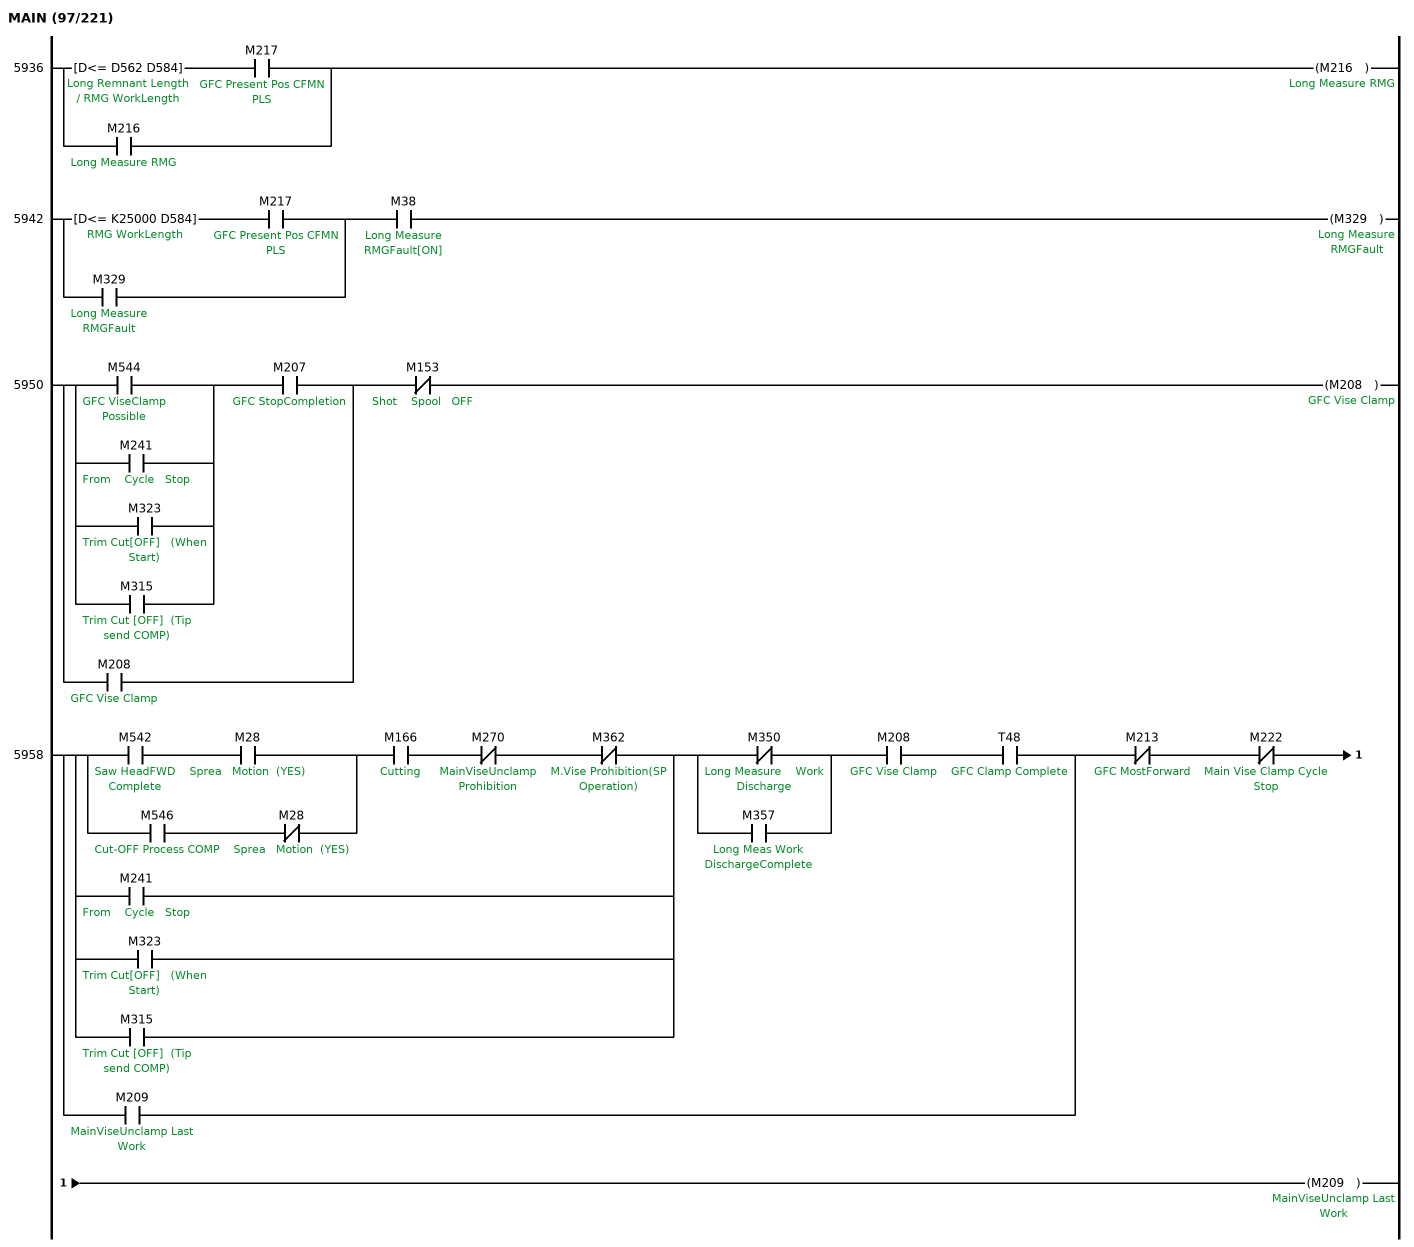
[picture p96: ladder of MAIN, rungs at steps 5936 to 5958]
5936  LDD<=   D562 D584  ; Long Remnant Length / RMG WorkLength
      AND     M217  ; GFC Present Pos CFMN PLS
      OR      M216  ; Long Measure RMG
      OUT     M216  ; Long Measure RMG
5942  LDD<=   K25000 D584  ; RMG WorkLength
      AND     M217  ; GFC Present Pos CFMN PLS
      OR      M329  ; Long Measure RMGFault
      AND     M38  ; Long Measure RMGFault[ON]
      OUT     M329  ; Long Measure RMGFault
5950  LD      M544  ; GFC ViseClamp   Possible
      OR      M241  ; From    Cycle   Stop
      OR      M323  ; Trim Cut[OFF]   (When   Start)
      OR      M315  ; Trim Cut [OFF]  (Tip send COMP)
      AND     M207  ; GFC StopCompletion
      OR      M208  ; GFC Vise Clamp
      ANI     M153  ; Shot    Spool   OFF
      OUT     M208  ; GFC Vise Clamp
5958  LD      M542  ; Saw HeadFWD     Complete
      AND     M28  ; Sprea   Motion  (YES)
      LD      M546  ; Cut-OFF Process COMP
      ANI     M28  ; Sprea   Motion  (YES)
      ORB
      AND     M166  ; Cutting
      ANI     M270  ; MainViseUnclamp Prohibition
      ANI     M362  ; M.Vise Prohibition(SP Operation)
      OR      M241  ; From    Cycle   Stop
      OR      M323  ; Trim Cut[OFF]   (When   Start)
      OR      M315  ; Trim Cut [OFF]  (Tip send COMP)
      LDI     M350  ; Long Measure    Work Discharge
      OR      M357  ; Long Meas Work DischargeComplete
      ANB
      AND     M208  ; GFC Vise Clamp
      AND     T48  ; GFC Clamp Complete
      OR      M209  ; MainViseUnclamp Last    Work
      ANI     M213  ; GFC MostForward
      ANI     M222  ; Main Vise Clamp Cycle Stop
      OUT     M209  ; MainViseUnclamp Last    Work
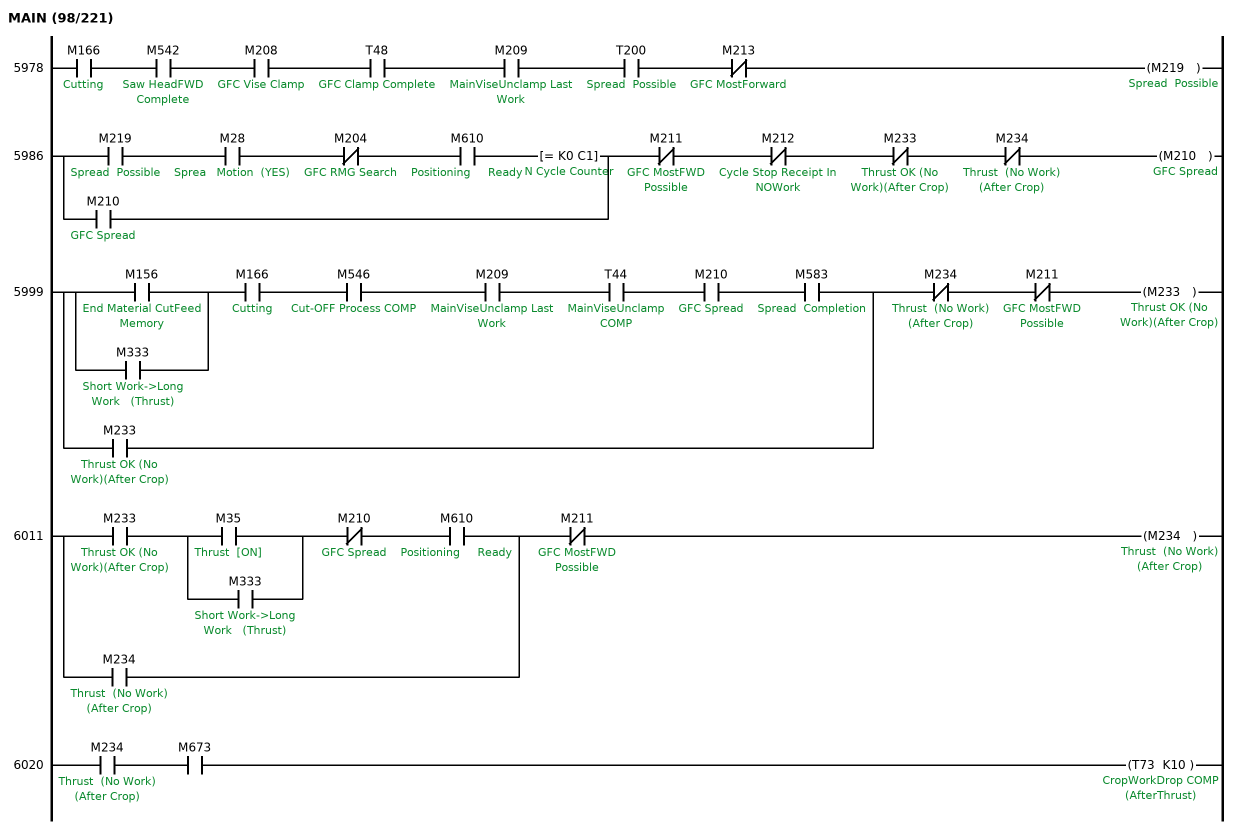
5978  LD      M166  ; Cutting
      AND     M542  ; Saw HeadFWD     Complete
      AND     M208  ; GFC Vise Clamp
      AND     T48  ; GFC Clamp Complete
      AND     M209  ; MainViseUnclamp Last    Work
      AND     T200  ; Spread  Possible
      ANI     M213  ; GFC MostForward
      OUT     M219  ; Spread  Possible
5986  LD      M219  ; Spread  Possible
      AND     M28  ; Sprea   Motion  (YES)
      ANI     M204  ; GFC RMG Search
      AND     M610  ; Positioning     Ready
      AND=    K0 C1  ; N Cycle Counter
      OR      M210  ; GFC Spread
      ANI     M211  ; GFC MostFWD     Possible
      ANI     M212  ; Cycle Stop Receipt In NOWork
      ANI     M233  ; Thrust OK (No Work)(After Crop)
      ANI     M234  ; Thrust  (No Work) (After Crop)
      OUT     M210  ; GFC Spread
5999  LD      M156  ; End Material CutFeed Memory
      OR      M333  ; Short Work->Long Work   (Thrust)
      AND     M166  ; Cutting
      AND     M546  ; Cut-OFF Process COMP
      AND     M209  ; MainViseUnclamp Last    Work
      AND     T44  ; MainViseUnclamp COMP
      AND     M210  ; GFC Spread
      AND     M583  ; Spread  Completion
      OR      M233  ; Thrust OK (No Work)(After Crop)
      ANI     M234  ; Thrust  (No Work) (After Crop)
      ANI     M211  ; GFC MostFWD     Possible
      OUT     M233  ; Thrust OK (No Work)(After Crop)
6011  LD      M233  ; Thrust OK (No Work)(After Crop)
      LD      M35  ; Thrust  [ON]
      OR      M333  ; Short Work->Long Work   (Thrust)
      ANB
      ANI     M210  ; GFC Spread
      AND     M610  ; Positioning     Ready
      OR      M234  ; Thrust  (No Work) (After Crop)
      ANI     M211  ; GFC MostFWD     Possible
      OUT     M234  ; Thrust  (No Work) (After Crop)
6020  LD      M234  ; Thrust  (No Work) (After Crop)
      AND     M673
      OUT     T73 K10  ; CropWorkDrop COMP (AfterThrust)
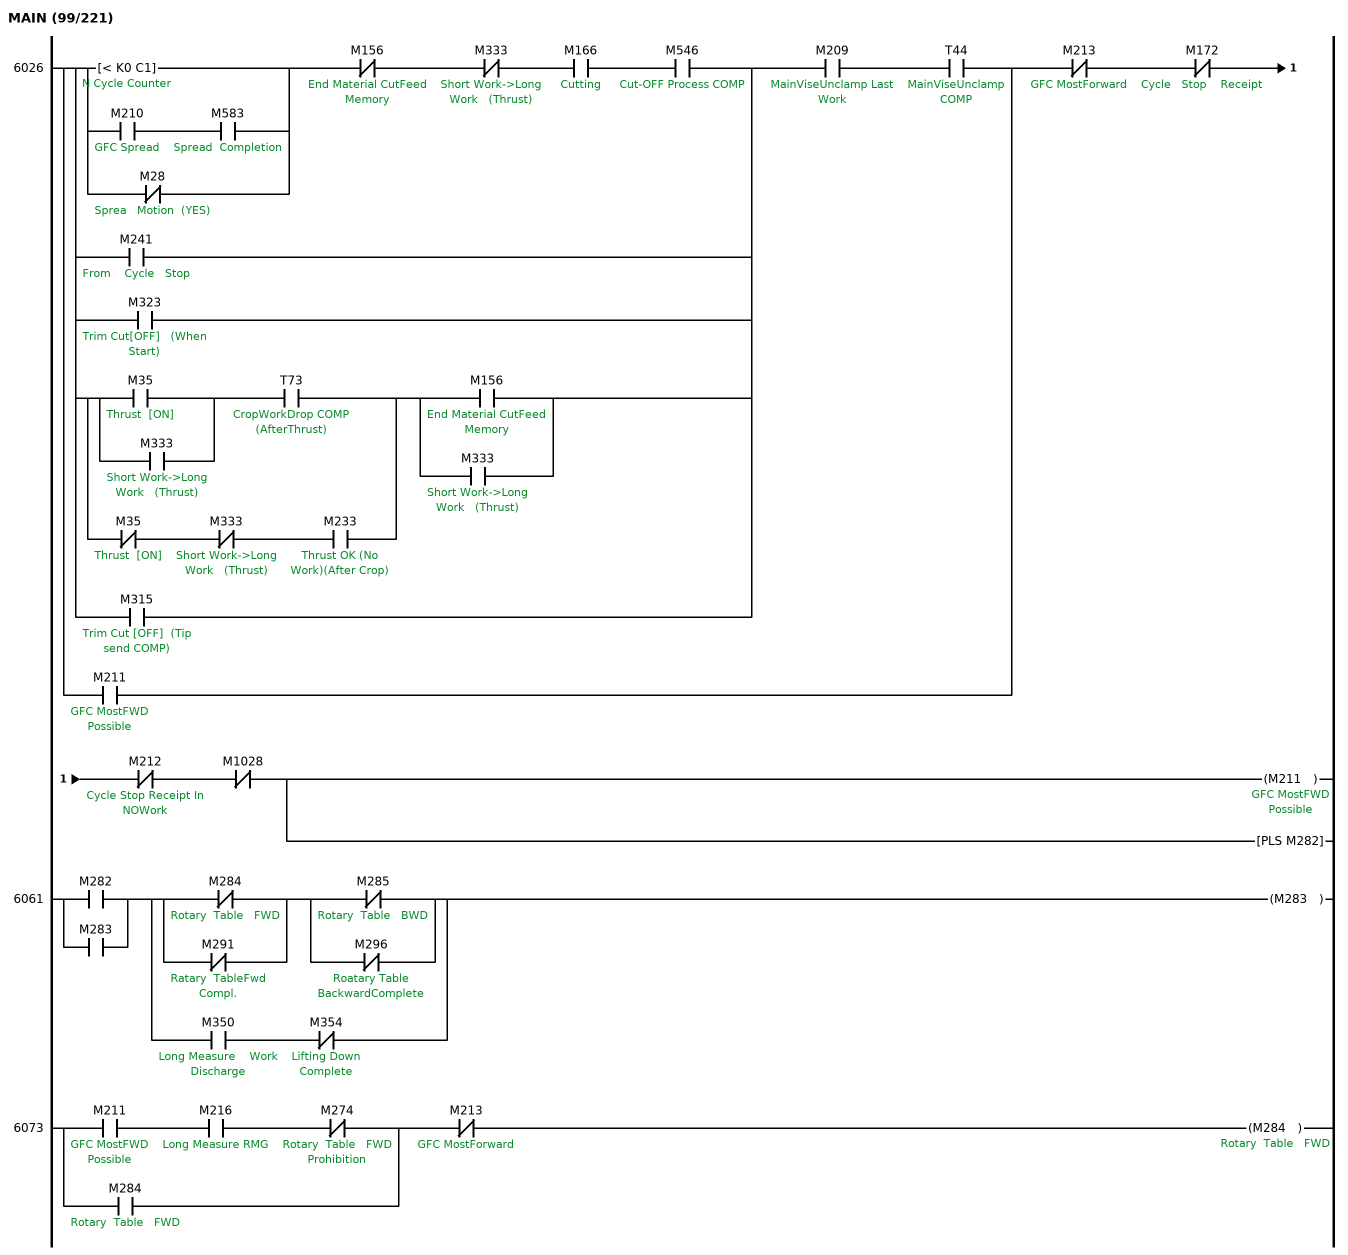
6026  LD<     K0 C1  ; N Cycle Counter
      LD      M210  ; GFC Spread
      AND     M583  ; Spread  Completion
      ORB
      ORI     M28  ; Sprea   Motion  (YES)
      ANI     M156  ; End Material CutFeed Memory
      ANI     M333  ; Short Work->Long Work   (Thrust)
      AND     M166  ; Cutting
      AND     M546  ; Cut-OFF Process COMP
      OR      M241  ; From    Cycle   Stop
      OR      M323  ; Trim Cut[OFF]   (When   Start)
      LD      M35  ; Thrust  [ON]
      OR      M333  ; Short Work->Long Work   (Thrust)
      AND     T73  ; CropWorkDrop COMP (AfterThrust)
      LDI     M35  ; Thrust  [ON]
      ANI     M333  ; Short Work->Long Work   (Thrust)
      AND     M233  ; Thrust OK (No Work)(After Crop)
      ORB
      LD      M156  ; End Material CutFeed Memory
      OR      M333  ; Short Work->Long Work   (Thrust)
      ANB
      ORB
      OR      M315  ; Trim Cut [OFF]  (Tip send COMP)
      AND     M209  ; MainViseUnclamp Last    Work
      AND     T44  ; MainViseUnclamp COMP
      OR      M211  ; GFC MostFWD     Possible
      ANI     M213  ; GFC MostForward
      ANI     M172  ; Cycle   Stop    Receipt
      ANI     M212  ; Cycle Stop Receipt In NOWork
      ANI     M1028
      OUT     M211  ; GFC MostFWD     Possible
      PLS     M282
6061  LD      M282
      OR      M283
      LDI     M284  ; Rotary  Table   FWD
      ORI     M291  ; Ratary  TableFwd Compl.
      LDI     M285  ; Rotary  Table   BWD
      ORI     M296  ; Roatary Table   BackwardComplete
      ANB
      LD      M350  ; Long Measure    Work Discharge
      ANI     M354  ; Lifting Down    Complete
      ORB
      ANB
      OUT     M283
6073  LD      M211  ; GFC MostFWD     Possible
      AND     M216  ; Long Measure RMG
      ANI     M274  ; Rotary  Table   FWD Prohibition
      OR      M284  ; Rotary  Table   FWD
      ANI     M213  ; GFC MostForward
      OUT     M284  ; Rotary  Table   FWD
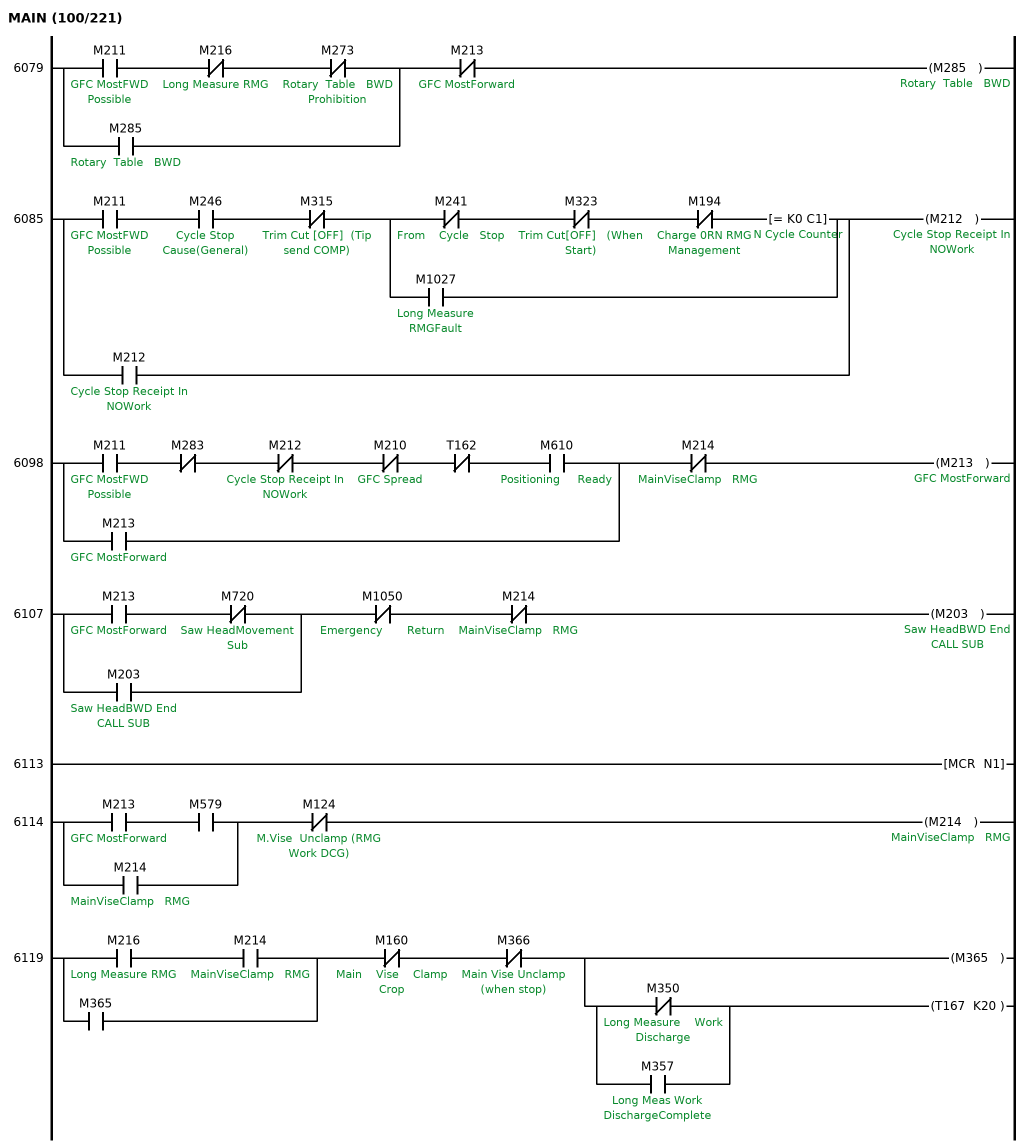
6079  LD      M211  ; GFC MostFWD     Possible
      ANI     M216  ; Long Measure RMG
      ANI     M273  ; Rotary  Table   BWD Prohibition
      OR      M285  ; Rotary  Table   BWD
      ANI     M213  ; GFC MostForward
      OUT     M285  ; Rotary  Table   BWD
6085  LD      M211  ; GFC MostFWD     Possible
      AND     M246  ; Cycle Stop Cause(General)
      ANI     M315  ; Trim Cut [OFF]  (Tip send COMP)
      LDI     M241  ; From    Cycle   Stop
      ANI     M323  ; Trim Cut[OFF]   (When   Start)
      ANI     M194  ; Charge 0RN RMG  Management
      AND=    K0 C1  ; N Cycle Counter
      OR      M1027  ; Long Measure RMGFault
      ANB
      OR      M212  ; Cycle Stop Receipt In NOWork
      OUT     M212  ; Cycle Stop Receipt In NOWork
6098  LD      M211  ; GFC MostFWD     Possible
      ANI     M283
      ANI     M212  ; Cycle Stop Receipt In NOWork
      ANI     M210  ; GFC Spread
      ANI     T162
      AND     M610  ; Positioning     Ready
      OR      M213  ; GFC MostForward
      ANI     M214  ; MainViseClamp   RMG
      OUT     M213  ; GFC MostForward
6107  LD      M213  ; GFC MostForward
      ANI     M720  ; Saw HeadMovementSub
      OR      M203  ; Saw HeadBWD End CALL SUB
      ANI     M1050  ; Emergency       Return
      ANI     M214  ; MainViseClamp   RMG
      OUT     M203  ; Saw HeadBWD End CALL SUB
6113  MCR     N1
6114  LD      M213  ; GFC MostForward
      AND     M579
      OR      M214  ; MainViseClamp   RMG
      ANI     M124  ; M.Vise  Unclamp (RMG Work DCG)
      OUT     M214  ; MainViseClamp   RMG
6119  LD      M216  ; Long Measure RMG
      AND     M214  ; MainViseClamp   RMG
      OR      M365
      ANI     M160  ; Main    Vise    Clamp   Crop
      ANI     M366  ; Main Vise Unclamp (when stop)
      OUT     M365
      LDI     M350  ; Long Measure    Work Discharge
      OR      M357  ; Long Meas Work DischargeComplete
      ANB
      OUT     T167 K20
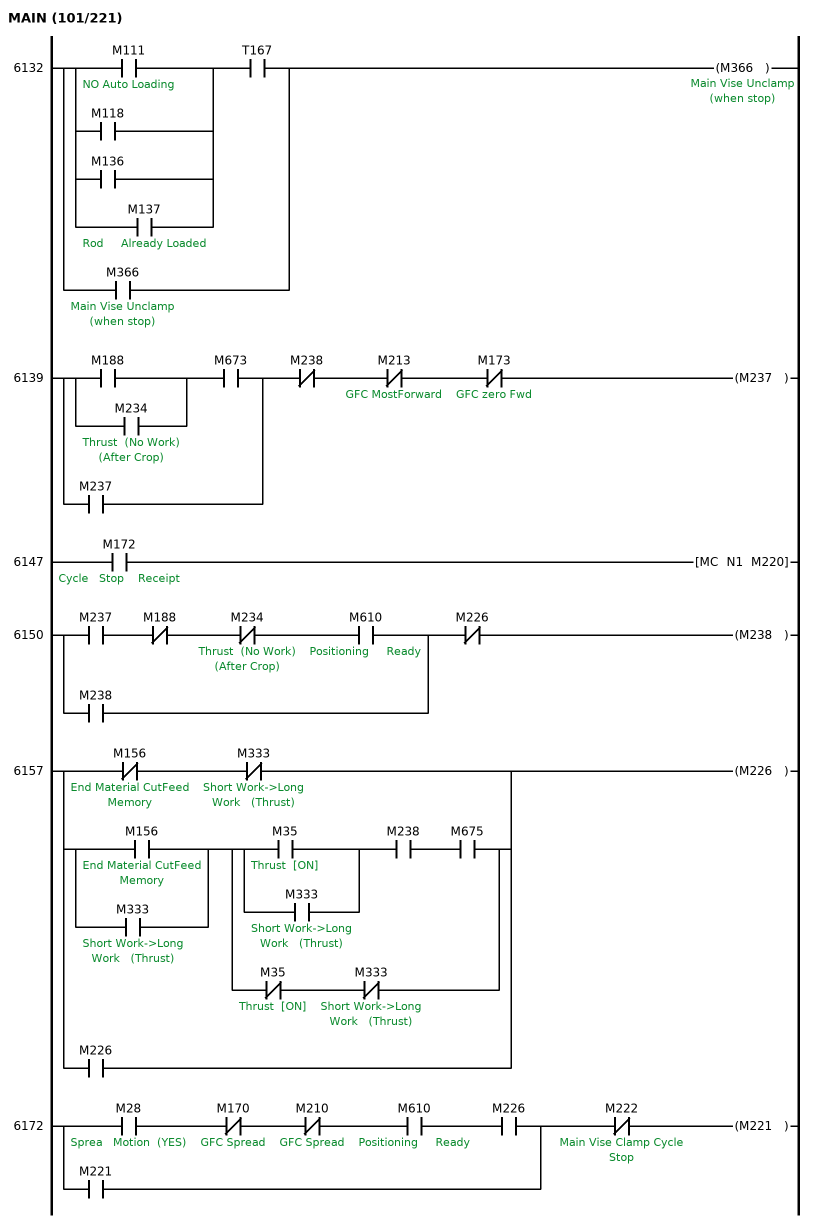
6132  LD      M111  ; NO Auto Loading
      OR      M118
      OR      M136
      OR      M137  ; Rod     Already Loaded
      AND     T167
      OR      M366  ; Main Vise Unclamp (when stop)
      OUT     M366  ; Main Vise Unclamp (when stop)
6139  LD      M188
      OR      M234  ; Thrust  (No Work) (After Crop)
      AND     M673
      OR      M237
      ANI     M238
      ANI     M213  ; GFC MostForward
      ANI     M173  ; GFC zero Fwd
      OUT     M237
6147  LD      M172  ; Cycle   Stop    Receipt
      MC      N1 M220
6150  LD      M237
      ANI     M188
      ANI     M234  ; Thrust  (No Work) (After Crop)
      AND     M610  ; Positioning     Ready
      OR      M238
      ANI     M226
      OUT     M238
6157  LDI     M156  ; End Material CutFeed Memory
      ANI     M333  ; Short Work->Long Work   (Thrust)
      LD      M156  ; End Material CutFeed Memory
      OR      M333  ; Short Work->Long Work   (Thrust)
      LD      M35  ; Thrust  [ON]
      OR      M333  ; Short Work->Long Work   (Thrust)
      AND     M238
      AND     M675
      LDI     M35  ; Thrust  [ON]
      ANI     M333  ; Short Work->Long Work   (Thrust)
      ORB
      ANB
      ORB
      OR      M226
      OUT     M226
6172  LD      M28  ; Sprea   Motion  (YES)
      ANI     M170  ; GFC Spread
      ANI     M210  ; GFC Spread
      AND     M610  ; Positioning     Ready
      AND     M226
      OR      M221
      ANI     M222  ; Main Vise Clamp Cycle Stop
      OUT     M221
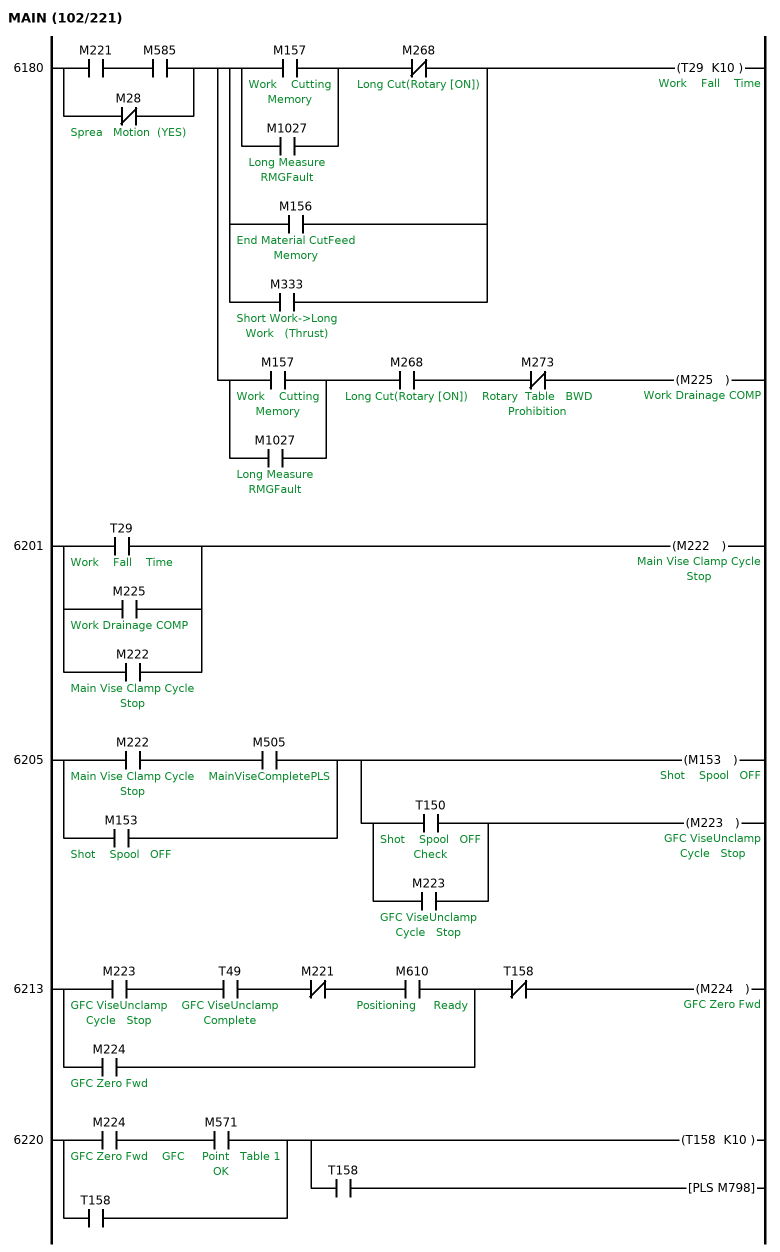
6180  LD      M221
      AND     M585
      ORI     M28  ; Sprea   Motion  (YES)
      MPS
      LD      M157  ; Work    Cutting Memory
      OR      M1027  ; Long Measure RMGFault
      ANI     M268  ; Long Cut(Rotary [ON])
      OR      M156  ; End Material CutFeed Memory
      OR      M333  ; Short Work->Long Work   (Thrust)
      ANB
      OUT     T29 K10  ; Work    Fall    Time
      MPP
      LD      M157  ; Work    Cutting Memory
      OR      M1027  ; Long Measure RMGFault
      ANB
      AND     M268  ; Long Cut(Rotary [ON])
      ANI     M273  ; Rotary  Table   BWD Prohibition
      OUT     M225  ; Work Drainage COMP
6201  LD      T29  ; Work    Fall    Time
      OR      M225  ; Work Drainage COMP
      OR      M222  ; Main Vise Clamp Cycle Stop
      OUT     M222  ; Main Vise Clamp Cycle Stop
6205  LD      M222  ; Main Vise Clamp Cycle Stop
      AND     M505  ; MainViseCompletePLS
      OR      M153  ; Shot    Spool   OFF
      OUT     M153  ; Shot    Spool   OFF
      LD      T150  ; Shot    Spool   OFF     Check
      OR      M223  ; GFC ViseUnclamp Cycle   Stop
      ANB
      OUT     M223  ; GFC ViseUnclamp Cycle   Stop
6213  LD      M223  ; GFC ViseUnclamp Cycle   Stop
      AND     T49  ; GFC ViseUnclamp Complete
      ANI     M221
      AND     M610  ; Positioning     Ready
      OR      M224  ; GFC Zero Fwd
      ANI     T158
      OUT     M224  ; GFC Zero Fwd
6220  LD      M224  ; GFC Zero Fwd
      AND     M571  ; GFC     Point   Table 1 OK
      OR      T158
      OUT     T158 K10
      AND     T158
      PLS     M798
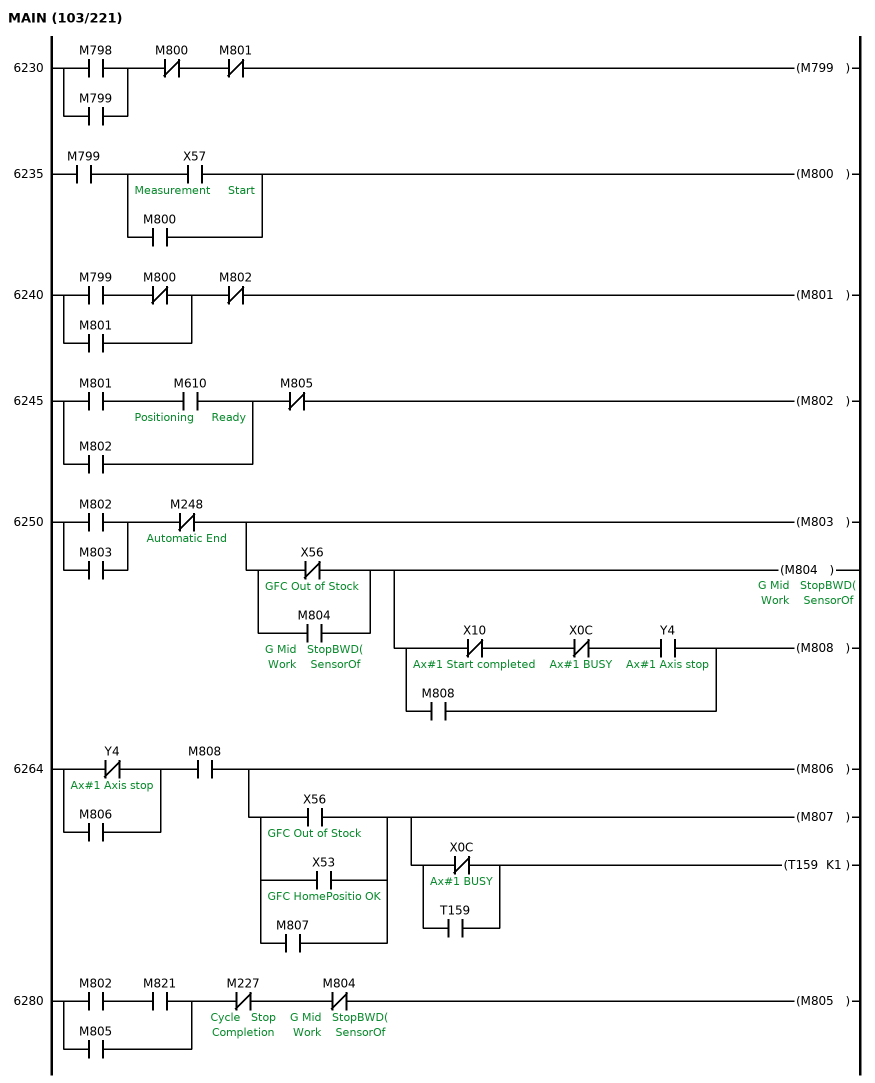
6230  LD      M798
      OR      M799
      ANI     M800
      ANI     M801
      OUT     M799
6235  LD      M799
      LD      X57  ; Measurement     Start
      OR      M800
      ANB
      OUT     M800
6240  LD      M799
      ANI     M800
      OR      M801
      ANI     M802
      OUT     M801
6245  LD      M801
      AND     M610  ; Positioning     Ready
      OR      M802
      ANI     M805
      OUT     M802
6250  LD      M802
      OR      M803
      ANI     M248  ; Automatic End
      OUT     M803
      LDI     X56  ; GFC Out of Stock
      OR      M804  ; G Mid   StopBWD(Work    SensorOf
      ANB
      OUT     M804  ; G Mid   StopBWD(Work    SensorOf
      LDI     X10  ; Ax#1 Start completed
      ANI     X0C  ; Ax#1 BUSY
      AND     Y4  ; Ax#1 Axis stop
      OR      M808
      ANB
      OUT     M808
6264  LDI     Y4  ; Ax#1 Axis stop
      OR      M806
      AND     M808
      OUT     M806
      LD      X56  ; GFC Out of Stock
      OR      X53  ; GFC HomePositio OK
      OR      M807
      ANB
      OUT     M807
      LDI     X0C  ; Ax#1 BUSY
      OR      T159
      ANB
      OUT     T159 K1
6280  LD      M802
      AND     M821
      OR      M805
      ANI     M227  ; Cycle   Stop    Completion
      ANI     M804  ; G Mid   StopBWD(Work    SensorOf
      OUT     M805
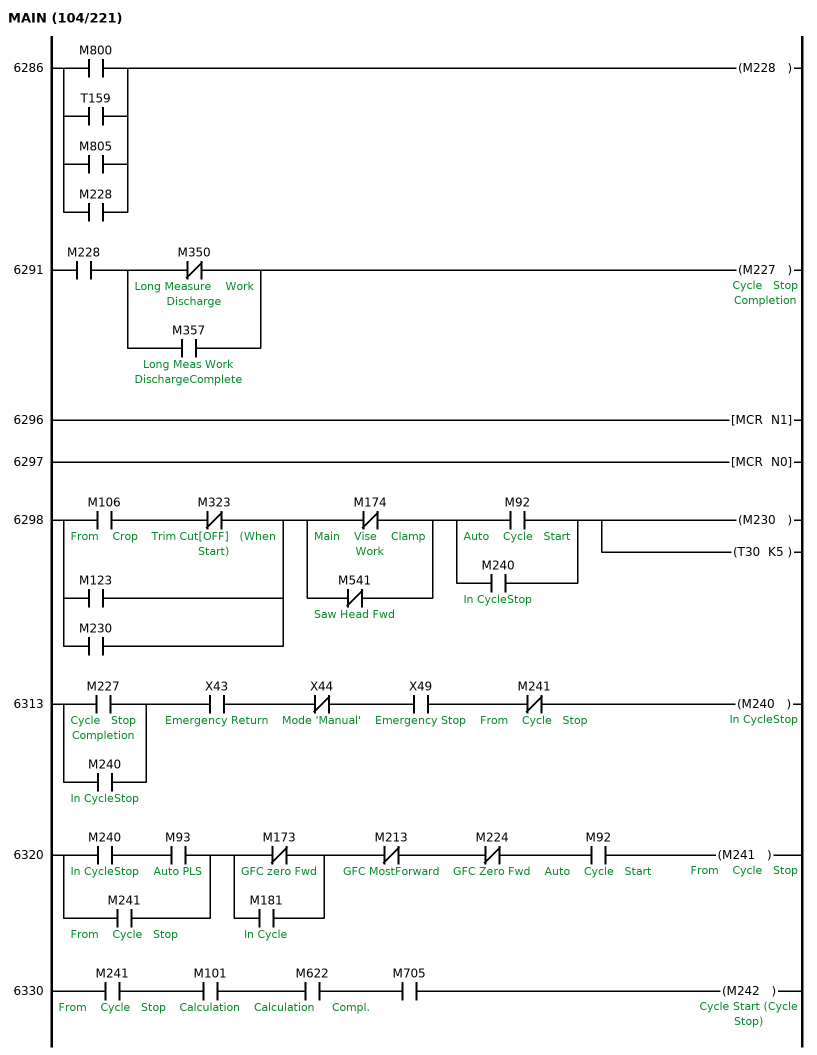
6286  LD      M800
      OR      T159
      OR      M805
      OR      M228
      OUT     M228
6291  LD      M228
      LDI     M350  ; Long Measure    Work Discharge
      OR      M357  ; Long Meas Work DischargeComplete
      ANB
      OUT     M227  ; Cycle   Stop    Completion
6296  MCR     N1
6297  MCR     N0
6298  LD      M106  ; From    Crop
      ANI     M323  ; Trim Cut[OFF]   (When   Start)
      OR      M123
      OR      M230
      LDI     M174  ; Main    Vise    Clamp   Work
      ORI     M541  ; Saw Head Fwd
      ANB
      LD      M92  ; Auto    Cycle   Start
      OR      M240  ; In CycleStop
      ANB
      OUT     M230
      OUT     T30 K5
6313  LD      M227  ; Cycle   Stop    Completion
      OR      M240  ; In CycleStop
      AND     X43  ; Emergency Return
      ANI     X44  ; Mode 'Manual'
      AND     X49  ; Emergency Stop
      ANI     M241  ; From    Cycle   Stop
      OUT     M240  ; In CycleStop
6320  LD      M240  ; In CycleStop
      AND     M93  ; Auto PLS
      OR      M241  ; From    Cycle   Stop
      LDI     M173  ; GFC zero Fwd
      OR      M181  ; In Cycle
      ANB
      ANI     M213  ; GFC MostForward
      ANI     M224  ; GFC Zero Fwd
      AND     M92  ; Auto    Cycle   Start
      OUT     M241  ; From    Cycle   Stop
6330  LD      M241  ; From    Cycle   Stop
      AND     M101  ; Calculation
      AND     M622  ; Calculation     Compl.
      AND     M705
      OUT     M242  ; Cycle Start (Cycle Stop)
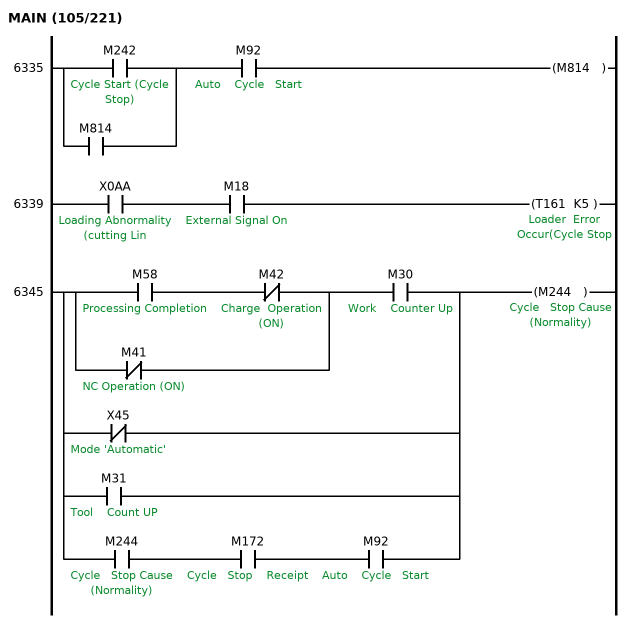
6335  LD      M242  ; Cycle Start (Cycle Stop)
      OR      M814
      AND     M92  ; Auto    Cycle   Start
      OUT     M814
6339  LD      X0AA  ; Loading Abnormality (cutting Lin
      AND     M18  ; External Signal On
      OUT     T161 K5  ; Loader  Error   Occur(Cycle Stop
6345  LD      M58  ; Processing Completion
      ANI     M42  ; Charge  Operation (ON)
      ORI     M41  ; NC Operation (ON)
      AND     M30  ; Work    Counter Up
      ORI     X45  ; Mode 'Automatic'
      OR      M31  ; Tool    Count UP
      LD      M244  ; Cycle   Stop Cause (Normality)
      AND     M172  ; Cycle   Stop    Receipt
      AND     M92  ; Auto    Cycle   Start
      ORB
      OUT     M244  ; Cycle   Stop Cause (Normality)
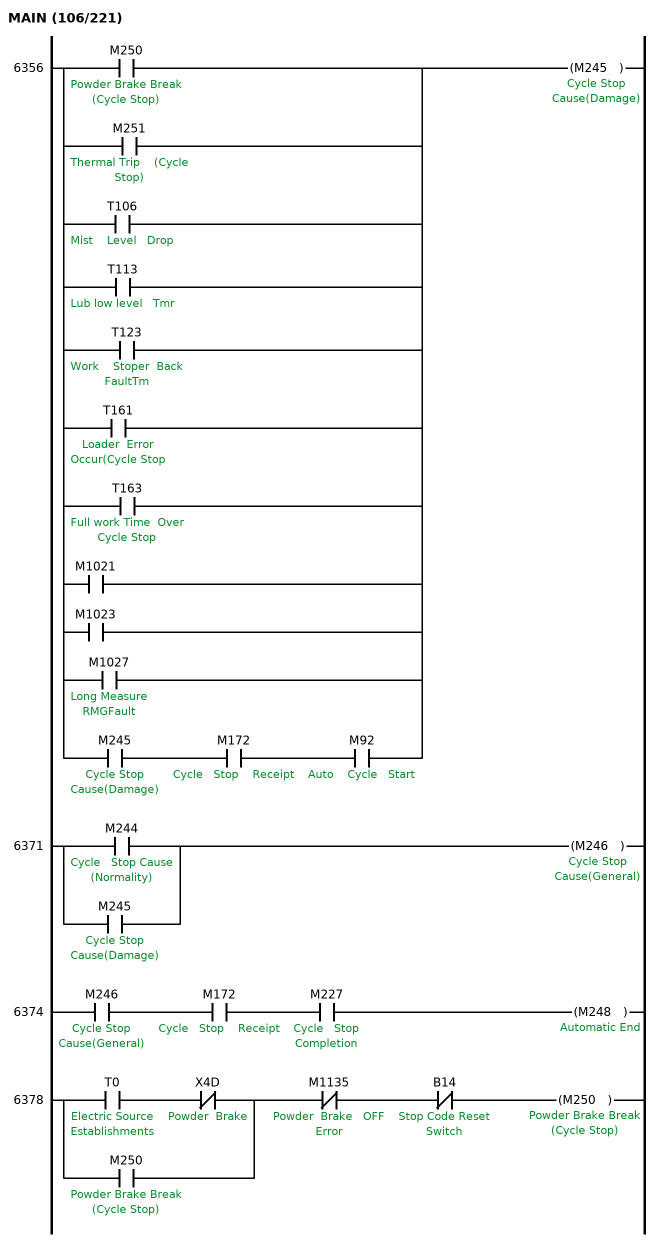
6356  LD      M250  ; Powder Brake Break (Cycle Stop)
      OR      M251  ; Thermal Trip    (Cycle  Stop)
      OR      T106  ; Mist    Level   Drop
      OR      T113  ; Lub low level   Tmr
      OR      T123  ; Work    Stoper  Back    FaultTm
      OR      T161  ; Loader  Error   Occur(Cycle Stop
      OR      T163  ; Full work Time  Over Cycle Stop
      OR      M1021
      OR      M1023
      OR      M1027  ; Long Measure RMGFault
      LD      M245  ; Cycle Stop Cause(Damage)
      AND     M172  ; Cycle   Stop    Receipt
      AND     M92  ; Auto    Cycle   Start
      ORB
      OUT     M245  ; Cycle Stop Cause(Damage)
6371  LD      M244  ; Cycle   Stop Cause (Normality)
      OR      M245  ; Cycle Stop Cause(Damage)
      OUT     M246  ; Cycle Stop Cause(General)
6374  LD      M246  ; Cycle Stop Cause(General)
      AND     M172  ; Cycle   Stop    Receipt
      AND     M227  ; Cycle   Stop    Completion
      OUT     M248  ; Automatic End
6378  LD      T0  ; Electric Source Establishments
      ANI     X4D  ; Powder  Brake
      OR      M250  ; Powder Brake Break (Cycle Stop)
      ANI     M1135  ; Powder  Brake   OFF     Error
      ANI     B14  ; Stop Code Reset Switch
      OUT     M250  ; Powder Brake Break (Cycle Stop)
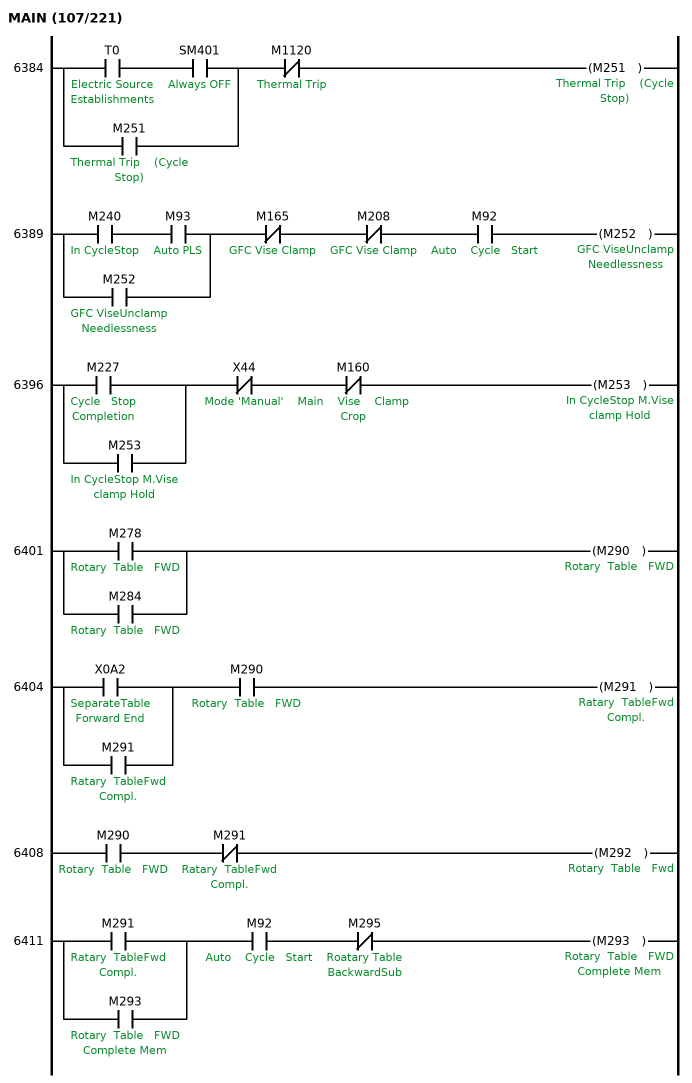
6384  LD      T0  ; Electric Source Establishments
      AND     SM401  ; Always OFF
      OR      M251  ; Thermal Trip    (Cycle  Stop)
      ANI     M1120  ; Thermal Trip
      OUT     M251  ; Thermal Trip    (Cycle  Stop)
6389  LD      M240  ; In CycleStop
      AND     M93  ; Auto PLS
      OR      M252  ; GFC ViseUnclamp Needlessness
      ANI     M165  ; GFC Vise Clamp
      ANI     M208  ; GFC Vise Clamp
      AND     M92  ; Auto    Cycle   Start
      OUT     M252  ; GFC ViseUnclamp Needlessness
6396  LD      M227  ; Cycle   Stop    Completion
      OR      M253  ; In CycleStop M.Vise clamp Hold
      ANI     X44  ; Mode 'Manual'
      ANI     M160  ; Main    Vise    Clamp   Crop
      OUT     M253  ; In CycleStop M.Vise clamp Hold
6401  LD      M278  ; Rotary  Table   FWD
      OR      M284  ; Rotary  Table   FWD
      OUT     M290  ; Rotary  Table   FWD
6404  LD      X0A2  ; SeparateTable   Forward End
      OR      M291  ; Ratary  TableFwd Compl.
      AND     M290  ; Rotary  Table   FWD
      OUT     M291  ; Ratary  TableFwd Compl.
6408  LD      M290  ; Rotary  Table   FWD
      ANI     M291  ; Ratary  TableFwd Compl.
      OUT     M292  ; Rotary  Table   Fwd
6411  LD      M291  ; Ratary  TableFwd Compl.
      OR      M293  ; Rotary  Table   FWD Complete Mem
      AND     M92  ; Auto    Cycle   Start
      ANI     M295  ; Roatary Table   BackwardSub
      OUT     M293  ; Rotary  Table   FWD Complete Mem
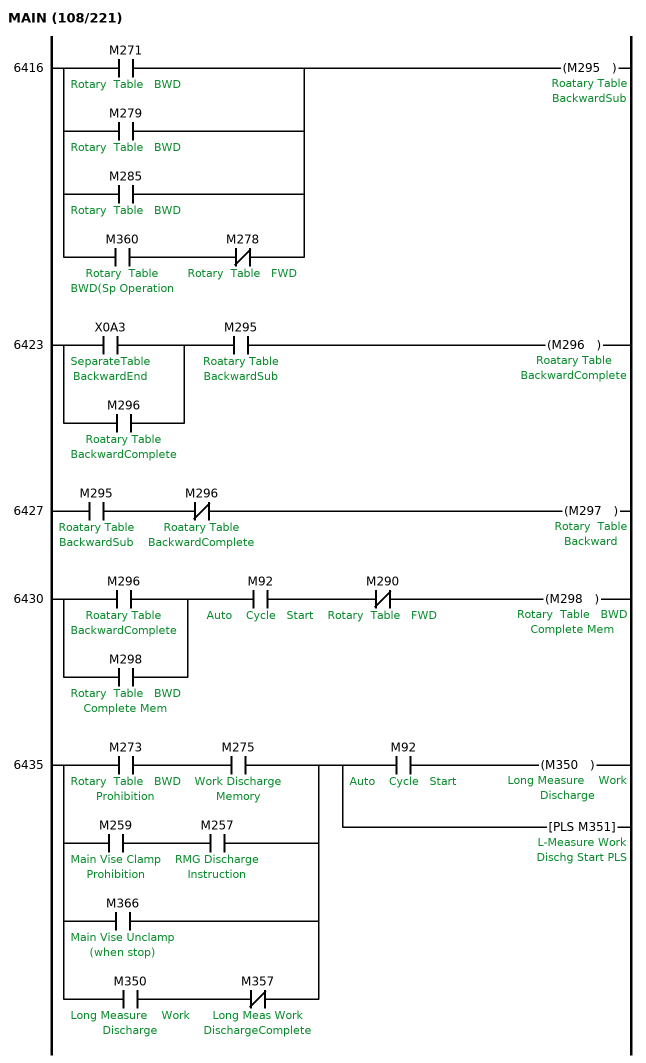
6416  LD      M271  ; Rotary  Table   BWD
      OR      M279  ; Rotary  Table   BWD
      OR      M285  ; Rotary  Table   BWD
      LD      M360  ; Rotary  Table   BWD(Sp Operation
      ANI     M278  ; Rotary  Table   FWD
      ORB
      OUT     M295  ; Roatary Table   BackwardSub
6423  LD      X0A3  ; SeparateTable   BackwardEnd
      OR      M296  ; Roatary Table   BackwardComplete
      AND     M295  ; Roatary Table   BackwardSub
      OUT     M296  ; Roatary Table   BackwardComplete
6427  LD      M295  ; Roatary Table   BackwardSub
      ANI     M296  ; Roatary Table   BackwardComplete
      OUT     M297  ; Rotary  Table   Backward
6430  LD      M296  ; Roatary Table   BackwardComplete
      OR      M298  ; Rotary  Table   BWD Complete Mem
      AND     M92  ; Auto    Cycle   Start
      ANI     M290  ; Rotary  Table   FWD
      OUT     M298  ; Rotary  Table   BWD Complete Mem
6435  LD      M273  ; Rotary  Table   BWD Prohibition
      AND     M275  ; Work Discharge  Memory
      LD      M259  ; Main Vise Clamp Prohibition
      AND     M257  ; RMG Discharge Instruction
      ORB
      OR      M366  ; Main Vise Unclamp (when stop)
      LD      M350  ; Long Measure    Work Discharge
      ANI     M357  ; Long Meas Work DischargeComplete
      ORB
      MPS
      AND     M92  ; Auto    Cycle   Start
      OUT     M350  ; Long Measure    Work Discharge
      MPP
      PLS     M351  ; L-Measure Work Dischg Start PLS
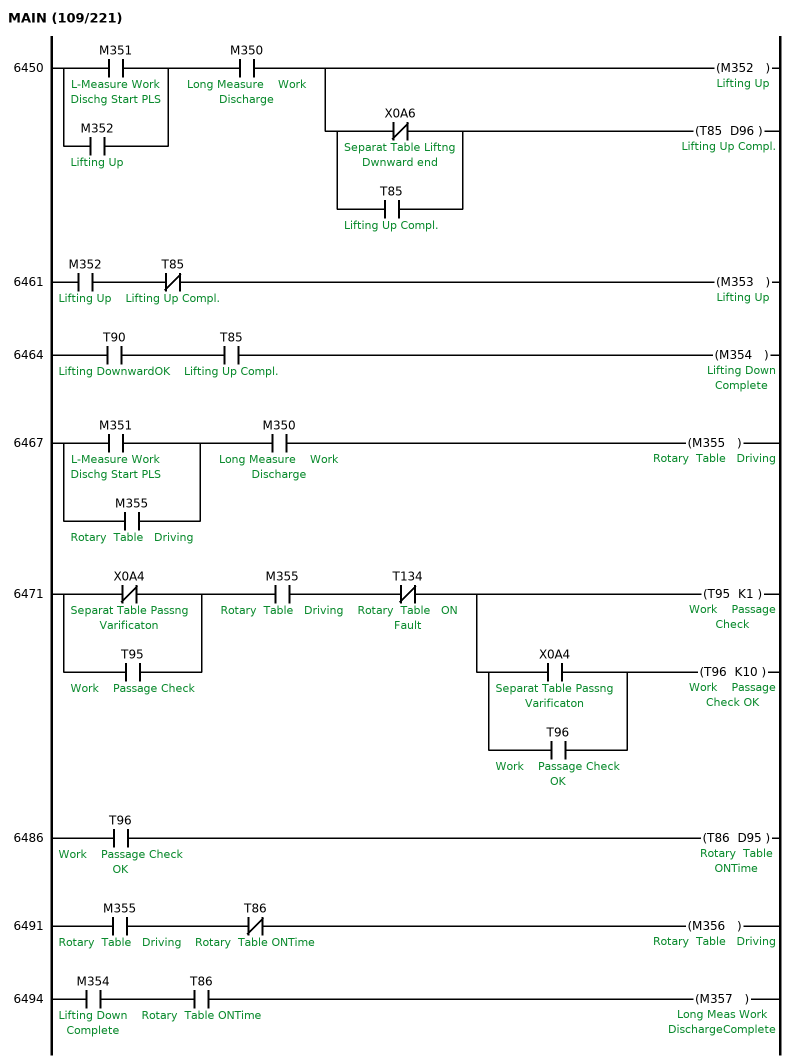
6450  LD      M351  ; L-Measure Work Dischg Start PLS
      OR      M352  ; Lifting Up
      AND     M350  ; Long Measure    Work Discharge
      OUT     M352  ; Lifting Up
      LDI     X0A6  ; Separat Table Liftng Dwnward end
      OR      T85  ; Lifting Up Compl.
      ANB
      OUT     T85 D96  ; Lifting Up Compl.
6461  LD      M352  ; Lifting Up
      ANI     T85  ; Lifting Up Compl.
      OUT     M353  ; Lifting Up
6464  LD      T90  ; Lifting DownwardOK
      AND     T85  ; Lifting Up Compl.
      OUT     M354  ; Lifting Down    Complete
6467  LD      M351  ; L-Measure Work Dischg Start PLS
      OR      M355  ; Rotary  Table   Driving
      AND     M350  ; Long Measure    Work Discharge
      OUT     M355  ; Rotary  Table   Driving
6471  LDI     X0A4  ; Separat Table Passng Varificaton
      OR      T95  ; Work    Passage Check
      AND     M355  ; Rotary  Table   Driving
      ANI     T134  ; Rotary  Table   ON Fault
      OUT     T95 K1  ; Work    Passage Check
      LD      X0A4  ; Separat Table Passng Varificaton
      OR      T96  ; Work    Passage Check OK
      ANB
      OUT     T96 K10  ; Work    Passage Check OK
6486  LD      T96  ; Work    Passage Check OK
      OUT     T86 D95  ; Rotary  Table ONTime
6491  LD      M355  ; Rotary  Table   Driving
      ANI     T86  ; Rotary  Table ONTime
      OUT     M356  ; Rotary  Table   Driving
6494  LD      M354  ; Lifting Down    Complete
      AND     T86  ; Rotary  Table ONTime
      OUT     M357  ; Long Meas Work DischargeComplete
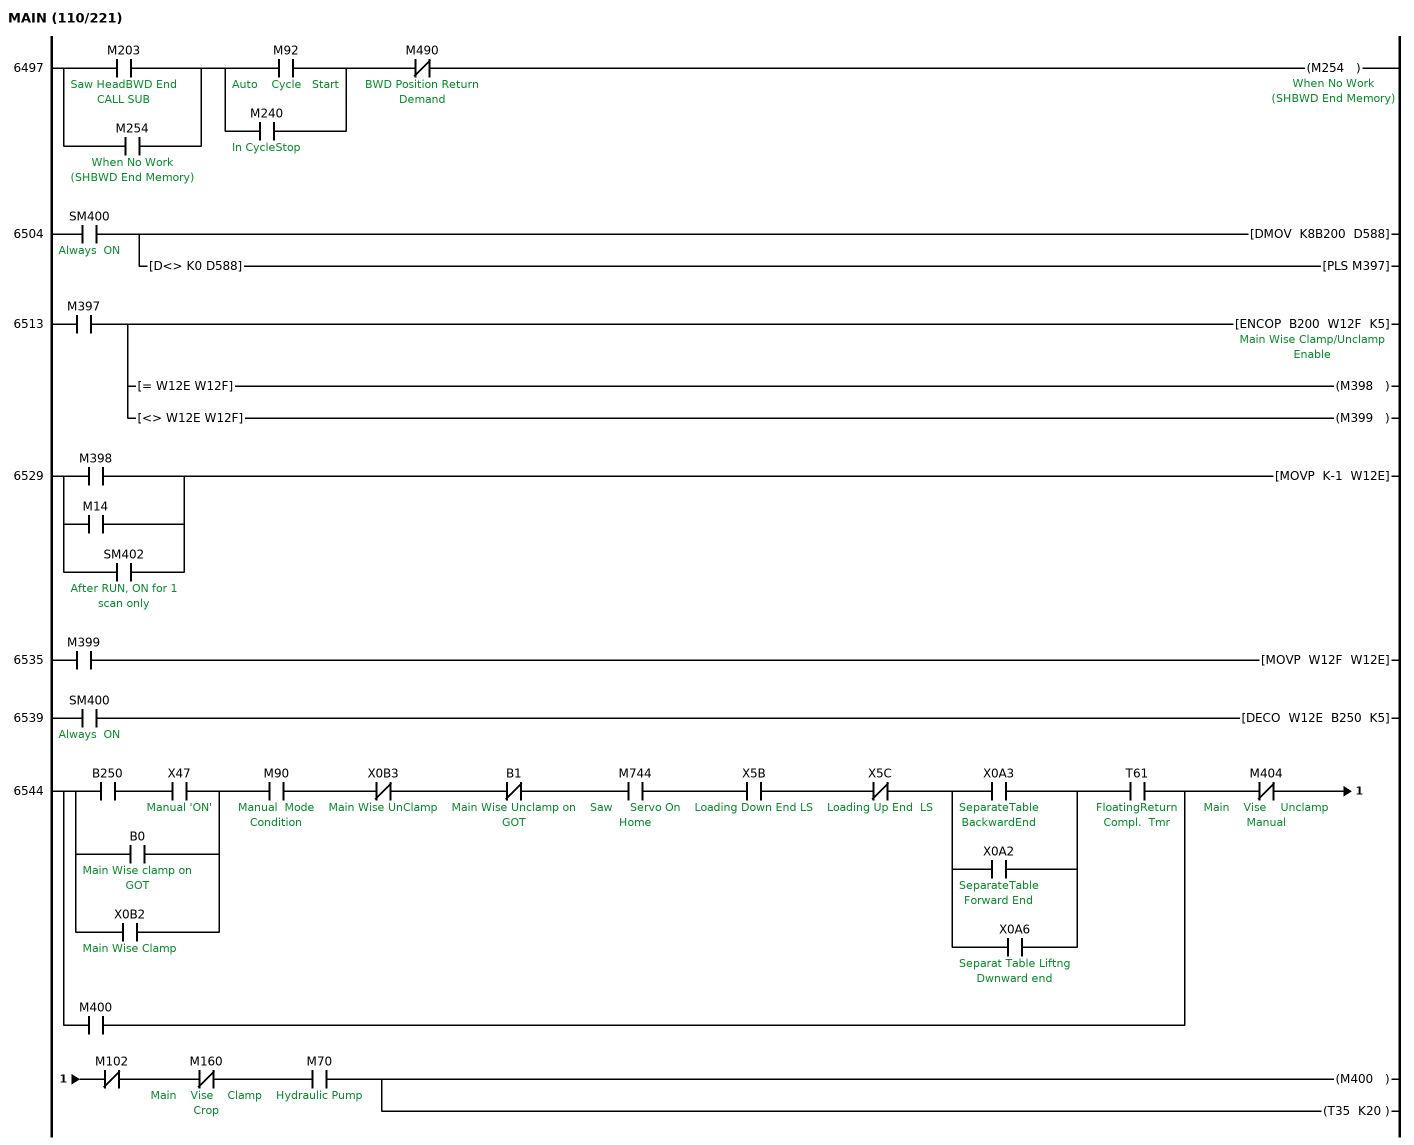
6497  LD      M203  ; Saw HeadBWD End CALL SUB
      OR      M254  ; When No Work (SHBWD End Memory)
      LD      M92  ; Auto    Cycle   Start
      OR      M240  ; In CycleStop
      ANB
      ANI     M490  ; BWD Position Return Demand
      OUT     M254  ; When No Work (SHBWD End Memory)
6504  LD      SM400  ; Always  ON
      DMOV    K8B200 D588  ; Main Wise Clamp/Unclamp Enable
      ANDD<>  K0 D588
      PLS     M397
6513  LD      M397
      ENCOP   B200 W12F K5
      MPS
      AND=    W12E W12F
      OUT     M398
      MPP
      AND<>   W12E W12F
      OUT     M399
6529  LD      M398
      OR      M14
      OR      SM402  ; After RUN, ON for 1 scan only
      MOVP    K-1 W12E
6535  LD      M399
      MOVP    W12F W12E
6539  LD      SM400  ; Always  ON
      DECO    W12E B250 K5
6544  LD      B250
      AND     X47  ; Manual 'ON'
      OR      B0  ; Main Wise clamp on GOT
      OR      X0B2  ; Main Wise Clamp
      AND     M90  ; Manual  Mode    Condition
      ANI     X0B3  ; Main Wise UnClamp
      ANI     B1  ; Main Wise Unclamp on GOT
      AND     M744  ; Saw     Servo On Home
      AND     X5B  ; Loading Down End LS
      ANI     X5C  ; Loading Up End  LS
      LD      X0A3  ; SeparateTable   BackwardEnd
      OR      X0A2  ; SeparateTable   Forward End
      OR      X0A6  ; Separat Table Liftng Dwnward end
      ANB
      AND     T61  ; FloatingReturn  Compl.  Tmr
      OR      M400
      ANI     M404  ; Main    Vise    Unclamp Manual
      ANI     M102
      ANI     M160  ; Main    Vise    Clamp   Crop
      AND     M70  ; Hydraulic Pump
      OUT     M400
      OUT     T35 K20
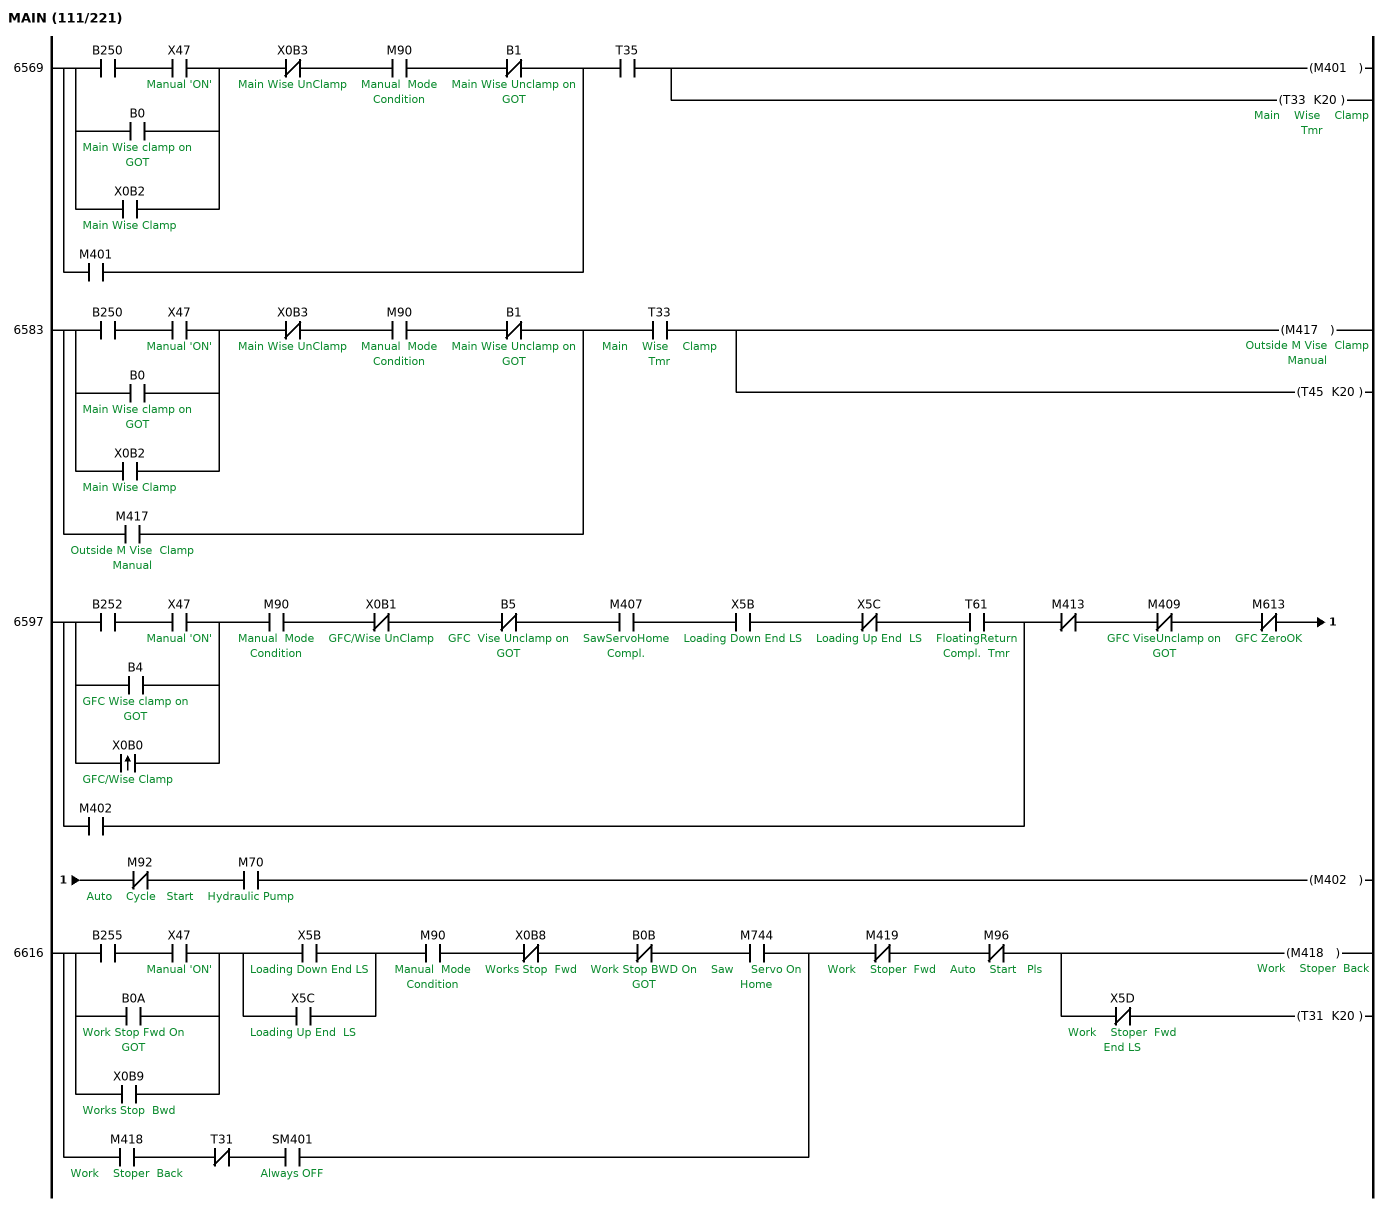
6569  LD      B250
      AND     X47  ; Manual 'ON'
      OR      B0  ; Main Wise clamp on GOT
      OR      X0B2  ; Main Wise Clamp
      ANI     X0B3  ; Main Wise UnClamp
      AND     M90  ; Manual  Mode    Condition
      ANI     B1  ; Main Wise Unclamp on GOT
      OR      M401
      AND     T35
      OUT     M401
      OUT     T33 K20  ; Main    Wise    Clamp   Tmr
6583  LD      B250
      AND     X47  ; Manual 'ON'
      OR      B0  ; Main Wise clamp on GOT
      OR      X0B2  ; Main Wise Clamp
      ANI     X0B3  ; Main Wise UnClamp
      AND     M90  ; Manual  Mode    Condition
      ANI     B1  ; Main Wise Unclamp on GOT
      OR      M417  ; Outside M Vise  Clamp   Manual
      AND     T33  ; Main    Wise    Clamp   Tmr
      OUT     M417  ; Outside M Vise  Clamp   Manual
      OUT     T45 K20
6597  LD      B252
      AND     X47  ; Manual 'ON'
      OR      B4  ; GFC Wise clamp on GOT
      ORP     X0B0  ; GFC/Wise Clamp
      AND     M90  ; Manual  Mode    Condition
      ANI     X0B1  ; GFC/Wise UnClamp
      ANI     B5  ; GFC  Vise Unclamp on GOT
      AND     M407  ; SawServoHome Compl.
      AND     X5B  ; Loading Down End LS
      ANI     X5C  ; Loading Up End  LS
      AND     T61  ; FloatingReturn  Compl.  Tmr
      OR      M402
      ANI     M413
      ANI     M409  ; GFC ViseUnclamp on GOT
      ANI     M613  ; GFC ZeroOK
      ANI     M92  ; Auto    Cycle   Start
      AND     M70  ; Hydraulic Pump
      OUT     M402
6616  LD      B255
      AND     X47  ; Manual 'ON'
      OR      B0A  ; Work Stop Fwd On GOT
      OR      X0B9  ; Works Stop  Bwd
      LD      X5B  ; Loading Down End LS
      OR      X5C  ; Loading Up End  LS
      ANB
      AND     M90  ; Manual  Mode    Condition
      ANI     X0B8  ; Works Stop  Fwd
      ANI     B0B  ; Work Stop BWD On GOT
      AND     M744  ; Saw     Servo On Home
      LD      M418  ; Work    Stoper  Back
      ANI     T31
      AND     SM401  ; Always OFF
      ORB
      ANI     M419  ; Work    Stoper  Fwd
      ANI     M96  ; Auto    Start   Pls
      OUT     M418  ; Work    Stoper  Back
      ANI     X5D  ; Work    Stoper  Fwd End LS
      OUT     T31 K20
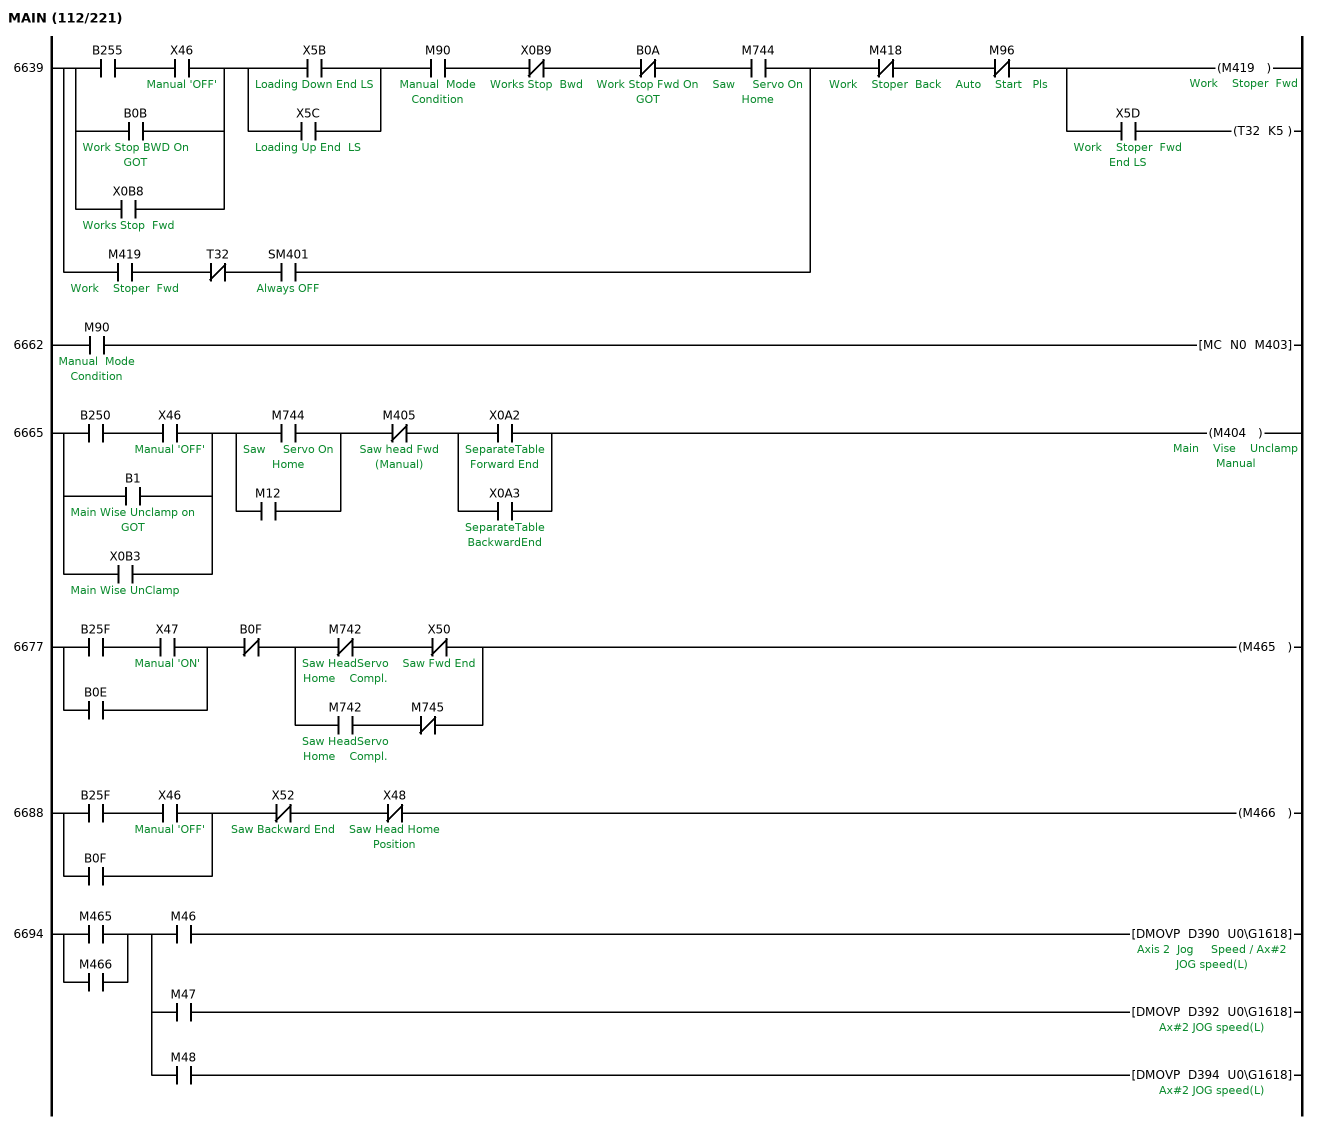
6639  LD      B255
      AND     X46  ; Manual 'OFF'
      OR      B0B  ; Work Stop BWD On GOT
      OR      X0B8  ; Works Stop  Fwd
      LD      X5B  ; Loading Down End LS
      OR      X5C  ; Loading Up End  LS
      ANB
      AND     M90  ; Manual  Mode    Condition
      ANI     X0B9  ; Works Stop  Bwd
      ANI     B0A  ; Work Stop Fwd On GOT
      AND     M744  ; Saw     Servo On Home
      LD      M419  ; Work    Stoper  Fwd
      ANI     T32
      AND     SM401  ; Always OFF
      ORB
      ANI     M418  ; Work    Stoper  Back
      ANI     M96  ; Auto    Start   Pls
      OUT     M419  ; Work    Stoper  Fwd
      AND     X5D  ; Work    Stoper  Fwd End LS
      OUT     T32 K5
6662  LD      M90  ; Manual  Mode    Condition
      MC      N0 M403
6665  LD      B250
      AND     X46  ; Manual 'OFF'
      OR      B1  ; Main Wise Unclamp on GOT
      OR      X0B3  ; Main Wise UnClamp
      LD      M744  ; Saw     Servo On Home
      OR      M12
      ANB
      ANI     M405  ; Saw head Fwd    (Manual)
      LD      X0A2  ; SeparateTable   Forward End
      OR      X0A3  ; SeparateTable   BackwardEnd
      ANB
      OUT     M404  ; Main    Vise    Unclamp Manual
6677  LD      B25F
      AND     X47  ; Manual 'ON'
      OR      B0E
      ANI     B0F
      LDI     M742  ; Saw HeadServo   Home    Compl.
      ANI     X50  ; Saw Fwd End
      LD      M742  ; Saw HeadServo   Home    Compl.
      ANI     M745
      ORB
      ANB
      OUT     M465
6688  LD      B25F
      AND     X46  ; Manual 'OFF'
      OR      B0F
      ANI     X52  ; Saw Backward End
      ANI     X48  ; Saw Head Home Position
      OUT     M466
6694  LD      M465
      OR      M466
      MPS
      AND     M46
      DMOVP   D390 U0\G1618
      MRD
      AND     M47
      DMOVP   D392 U0\G1618
      MPP
      AND     M48
      DMOVP   D394 U0\G1618
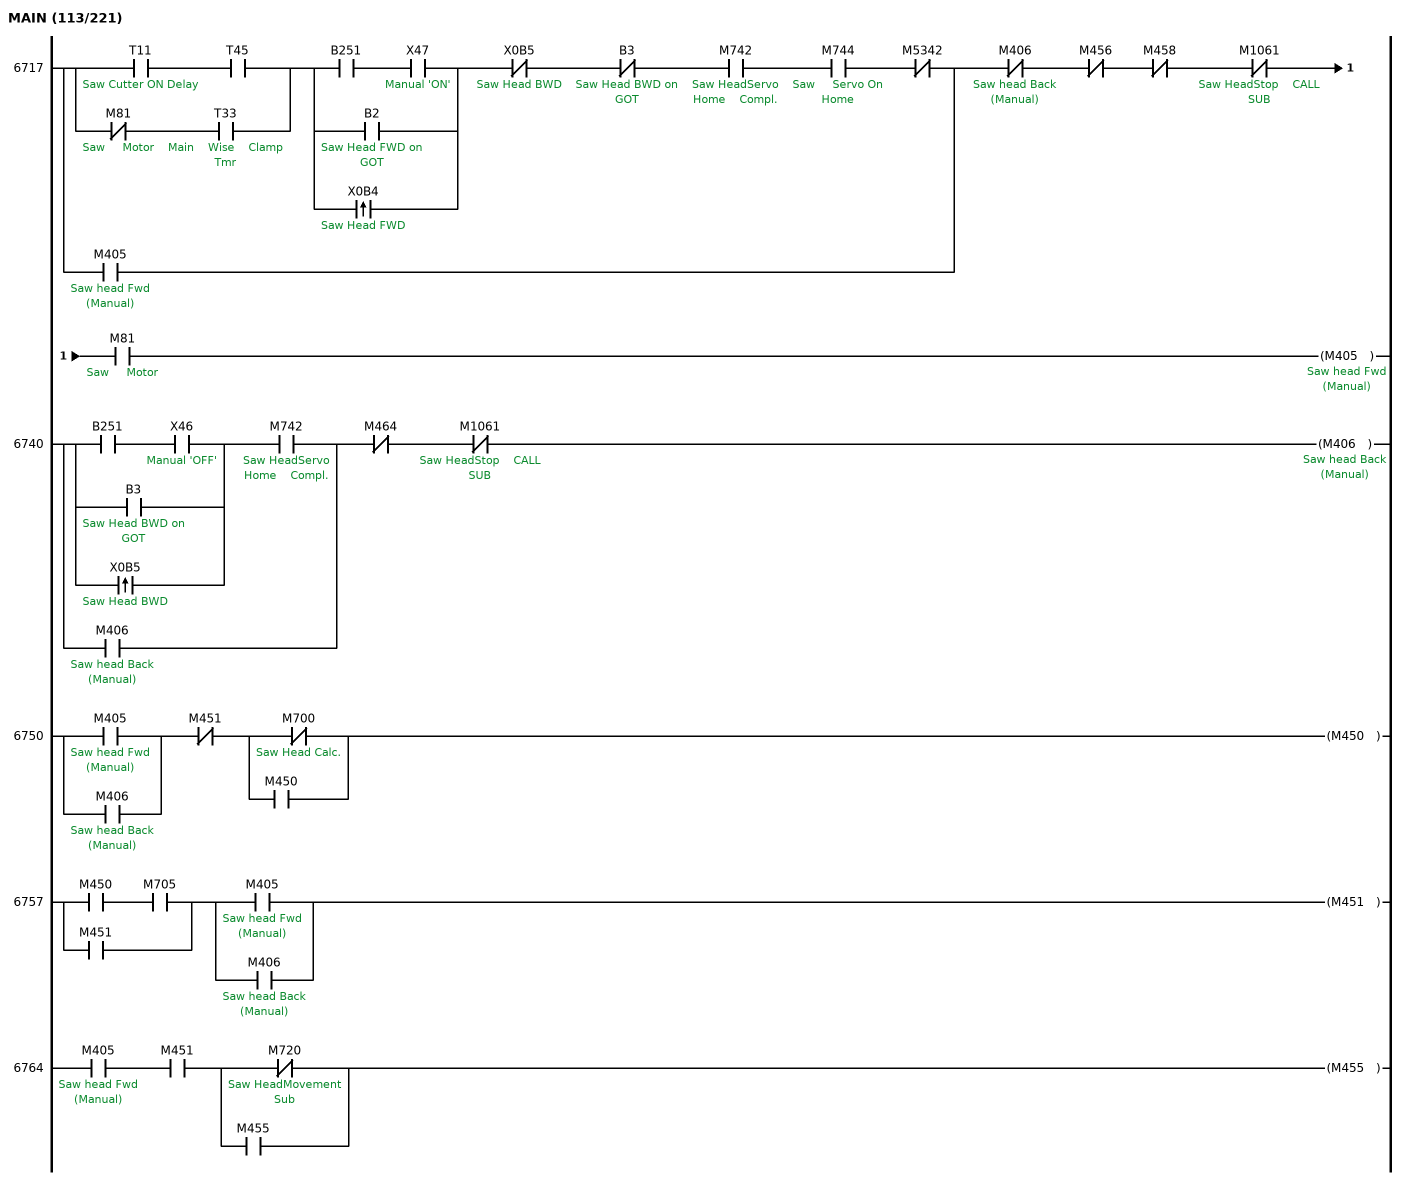
6717  LD      T11  ; Saw Cutter ON Delay
      AND     T45
      LDI     M81  ; Saw     Motor
      AND     T33  ; Main    Wise    Clamp   Tmr
      ORB
      LD      B251
      AND     X47  ; Manual 'ON'
      OR      B2  ; Saw Head FWD on GOT
      ORP     X0B4  ; Saw Head FWD
      ANB
      ANI     X0B5  ; Saw Head BWD
      ANI     B3  ; Saw Head BWD on GOT
      AND     M742  ; Saw HeadServo   Home    Compl.
      AND     M744  ; Saw     Servo On Home
      ANI     M5342
      OR      M405  ; Saw head Fwd    (Manual)
      ANI     M406  ; Saw head Back   (Manual)
      ANI     M456
      ANI     M458
      ANI     M1061  ; Saw HeadStop    CALL SUB
      AND     M81  ; Saw     Motor
      OUT     M405  ; Saw head Fwd    (Manual)
6740  LD      B251
      AND     X46  ; Manual 'OFF'
      OR      B3  ; Saw Head BWD on GOT
      ORP     X0B5  ; Saw Head BWD
      AND     M742  ; Saw HeadServo   Home    Compl.
      OR      M406  ; Saw head Back   (Manual)
      ANI     M464
      ANI     M1061  ; Saw HeadStop    CALL SUB
      OUT     M406  ; Saw head Back   (Manual)
6750  LD      M405  ; Saw head Fwd    (Manual)
      OR      M406  ; Saw head Back   (Manual)
      ANI     M451
      LDI     M700  ; Saw Head Calc.
      OR      M450
      ANB
      OUT     M450
6757  LD      M450
      AND     M705
      OR      M451
      LD      M405  ; Saw head Fwd    (Manual)
      OR      M406  ; Saw head Back   (Manual)
      ANB
      OUT     M451
6764  LD      M405  ; Saw head Fwd    (Manual)
      AND     M451
      LDI     M720  ; Saw HeadMovementSub
      OR      M455
      ANB
      OUT     M455
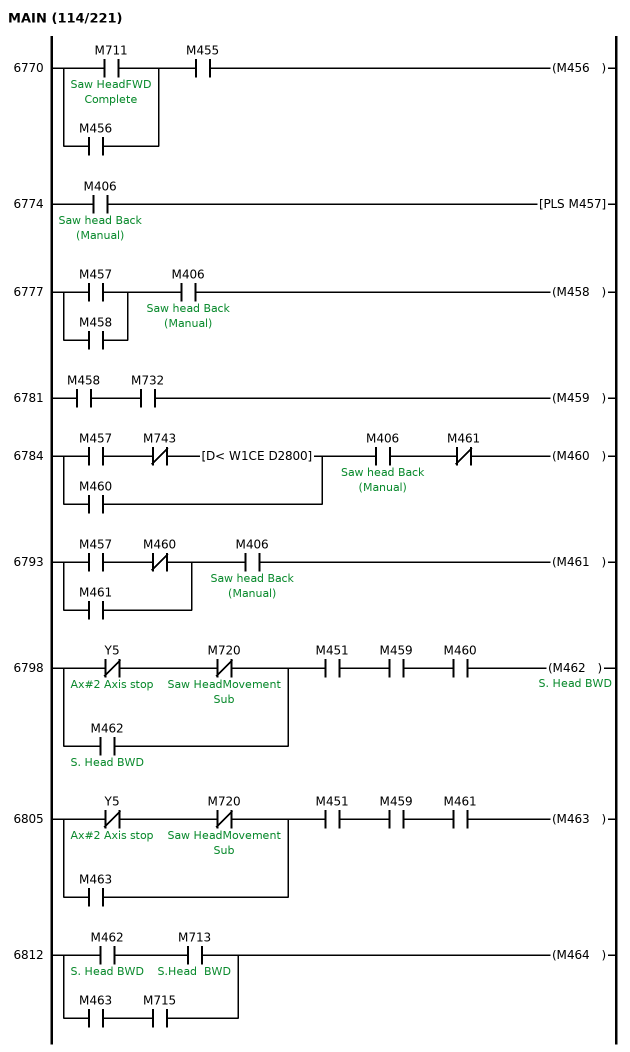
6770  LD      M711  ; Saw HeadFWD     Complete
      OR      M456
      AND     M455
      OUT     M456
6774  LD      M406  ; Saw head Back   (Manual)
      PLS     M457
6777  LD      M457
      OR      M458
      AND     M406  ; Saw head Back   (Manual)
      OUT     M458
6781  LD      M458
      AND     M732
      OUT     M459
6784  LD      M457
      ANI     M743
      ANDD<   W1CE D2800
      OR      M460
      AND     M406  ; Saw head Back   (Manual)
      ANI     M461
      OUT     M460
6793  LD      M457
      ANI     M460
      OR      M461
      AND     M406  ; Saw head Back   (Manual)
      OUT     M461
6798  LDI     Y5  ; Ax#2 Axis stop
      ANI     M720  ; Saw HeadMovementSub
      OR      M462  ; S. Head BWD
      AND     M451
      AND     M459
      AND     M460
      OUT     M462  ; S. Head BWD
6805  LDI     Y5  ; Ax#2 Axis stop
      ANI     M720  ; Saw HeadMovementSub
      OR      M463
      AND     M451
      AND     M459
      AND     M461
      OUT     M463
6812  LD      M462  ; S. Head BWD
      AND     M713  ; S.Head  BWD
      LD      M463
      AND     M715
      ORB
      OUT     M464
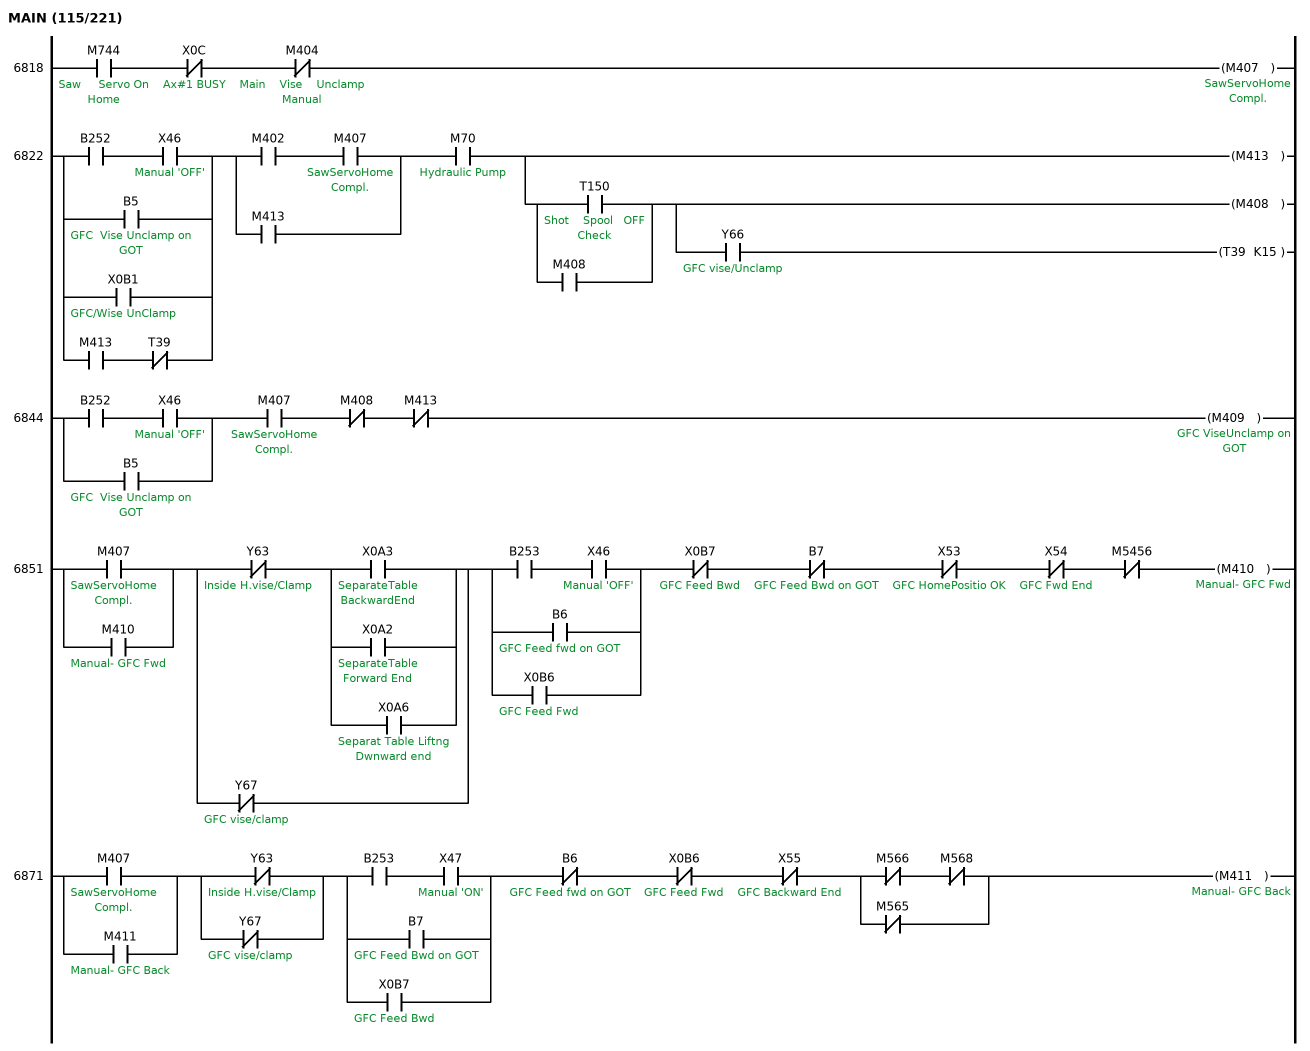
6818  LD      M744  ; Saw     Servo On Home
      ANI     X0C  ; Ax#1 BUSY
      ANI     M404  ; Main    Vise    Unclamp Manual
      OUT     M407  ; SawServoHome Compl.
6822  LD      B252
      AND     X46  ; Manual 'OFF'
      OR      B5  ; GFC  Vise Unclamp on GOT
      OR      X0B1  ; GFC/Wise UnClamp
      LD      M413
      ANI     T39
      ORB
      LD      M402
      AND     M407  ; SawServoHome Compl.
      OR      M413
      ANB
      AND     M70  ; Hydraulic Pump
      OUT     M413
      LD      T150  ; Shot    Spool   OFF     Check
      OR      M408
      ANB
      OUT     M408
      AND     Y66  ; GFC vise/Unclamp
      OUT     T39 K15
6844  LD      B252
      AND     X46  ; Manual 'OFF'
      OR      B5  ; GFC  Vise Unclamp on GOT
      AND     M407  ; SawServoHome Compl.
      ANI     M408
      ANI     M413
      OUT     M409  ; GFC ViseUnclamp on GOT
6851  LD      M407  ; SawServoHome Compl.
      OR      M410  ; Manual- GFC Fwd
      LDI     Y63  ; Inside H.vise/Clamp
      LD      X0A3  ; SeparateTable   BackwardEnd
      OR      X0A2  ; SeparateTable   Forward End
      OR      X0A6  ; Separat Table Liftng Dwnward end
      ANB
      ORI     Y67  ; GFC vise/clamp
      ANB
      LD      B253
      AND     X46  ; Manual 'OFF'
      OR      B6  ; GFC Feed fwd on GOT
      OR      X0B6  ; GFC Feed Fwd
      ANB
      ANI     X0B7  ; GFC Feed Bwd
      ANI     B7  ; GFC Feed Bwd on GOT
      ANI     X53  ; GFC HomePositio OK
      ANI     X54  ; GFC Fwd End
      ANI     M5456
      OUT     M410  ; Manual- GFC Fwd
6871  LD      M407  ; SawServoHome Compl.
      OR      M411  ; Manual- GFC Back
      LDI     Y63  ; Inside H.vise/Clamp
      ORI     Y67  ; GFC vise/clamp
      ANB
      LD      B253
      AND     X47  ; Manual 'ON'
      OR      B7  ; GFC Feed Bwd on GOT
      OR      X0B7  ; GFC Feed Bwd
      ANB
      ANI     B6  ; GFC Feed fwd on GOT
      ANI     X0B6  ; GFC Feed Fwd
      ANI     X55  ; GFC Backward End
      LDI     M566
      ANI     M568
      ORI     M565
      ANB
      OUT     M411  ; Manual- GFC Back
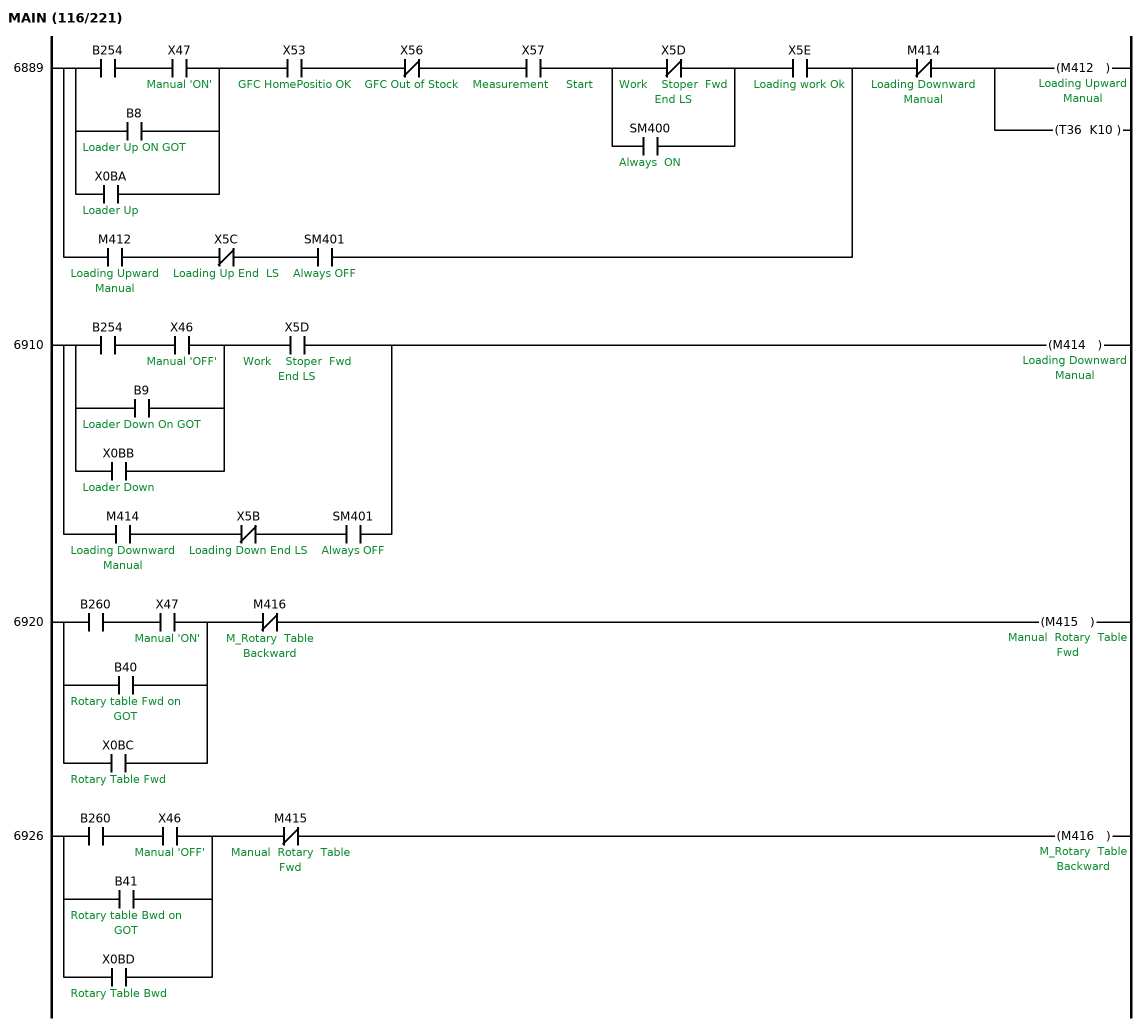
6889  LD      B254
      AND     X47  ; Manual 'ON'
      OR      B8  ; Loader Up ON GOT
      OR      X0BA  ; Loader Up
      AND     X53  ; GFC HomePositio OK
      ANI     X56  ; GFC Out of Stock
      AND     X57  ; Measurement     Start
      LDI     X5D  ; Work    Stoper  Fwd End LS
      OR      SM400  ; Always  ON
      ANB
      AND     X5E  ; Loading work Ok
      LD      M412  ; Loading Upward  Manual
      ANI     X5C  ; Loading Up End  LS
      AND     SM401  ; Always OFF
      ORB
      ANI     M414  ; Loading Downward Manual
      OUT     M412  ; Loading Upward  Manual
      OUT     T36 K10
6910  LD      B254
      AND     X46  ; Manual 'OFF'
      OR      B9  ; Loader Down On GOT
      OR      X0BB  ; Loader Down
      AND     X5D  ; Work    Stoper  Fwd End LS
      LD      M414  ; Loading Downward Manual
      ANI     X5B  ; Loading Down End LS
      AND     SM401  ; Always OFF
      ORB
      OUT     M414  ; Loading Downward Manual
6920  LD      B260
      AND     X47  ; Manual 'ON'
      OR      B40  ; Rotary table Fwd on GOT
      OR      X0BC  ; Rotary Table Fwd
      ANI     M416  ; M_Rotary  Table Backward
      OUT     M415  ; Manual  Rotary  Table   Fwd
6926  LD      B260
      AND     X46  ; Manual 'OFF'
      OR      B41  ; Rotary table Bwd on GOT
      OR      X0BD  ; Rotary Table Bwd
      ANI     M415  ; Manual  Rotary  Table   Fwd
      OUT     M416  ; M_Rotary  Table Backward
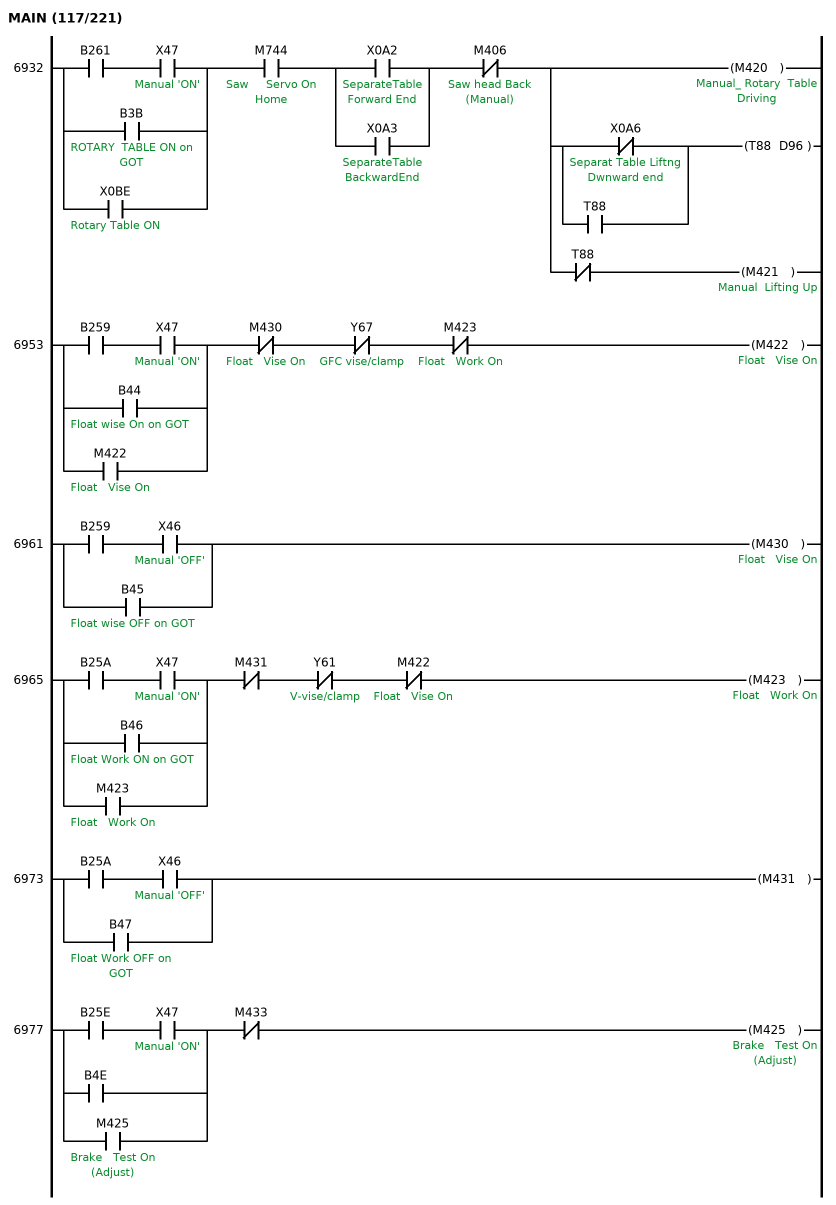
6932  LD      B261
      AND     X47  ; Manual 'ON'
      OR      B3B  ; ROTARY  TABLE ON on GOT
      OR      X0BE  ; Rotary Table ON
      AND     M744  ; Saw     Servo On Home
      LD      X0A2  ; SeparateTable   Forward End
      OR      X0A3  ; SeparateTable   BackwardEnd
      ANB
      ANI     M406  ; Saw head Back   (Manual)
      OUT     M420  ; Manual_ Rotary  Table   Driving
      MPS
      LDI     X0A6  ; Separat Table Liftng Dwnward end
      OR      T88
      ANB
      OUT     T88 D96
      MPP
      ANI     T88
      OUT     M421  ; Manual  Lifting Up
6953  LD      B259
      AND     X47  ; Manual 'ON'
      OR      B44  ; Float wise On on GOT
      OR      M422  ; Float   Vise On
      ANI     M430  ; Float   Vise On
      ANI     Y67  ; GFC vise/clamp
      ANI     M423  ; Float   Work On
      OUT     M422  ; Float   Vise On
6961  LD      B259
      AND     X46  ; Manual 'OFF'
      OR      B45  ; Float wise OFF on GOT
      OUT     M430  ; Float   Vise On
6965  LD      B25A
      AND     X47  ; Manual 'ON'
      OR      B46  ; Float Work ON on GOT
      OR      M423  ; Float   Work On
      ANI     M431
      ANI     Y61  ; V-vise/clamp
      ANI     M422  ; Float   Vise On
      OUT     M423  ; Float   Work On
6973  LD      B25A
      AND     X46  ; Manual 'OFF'
      OR      B47  ; Float Work OFF on GOT
      OUT     M431
6977  LD      B25E
      AND     X47  ; Manual 'ON'
      OR      B4E
      OR      M425  ; Brake   Test On (Adjust)
      ANI     M433
      OUT     M425  ; Brake   Test On (Adjust)
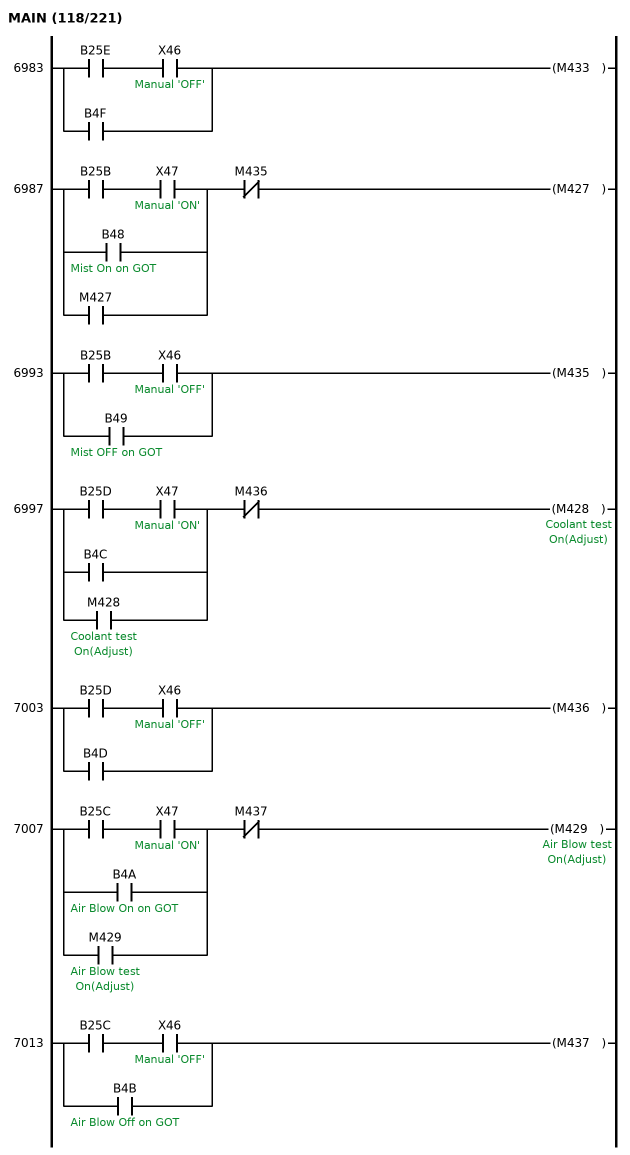
6983  LD      B25E
      AND     X46  ; Manual 'OFF'
      OR      B4F
      OUT     M433
6987  LD      B25B
      AND     X47  ; Manual 'ON'
      OR      B48  ; Mist On on GOT
      OR      M427
      ANI     M435
      OUT     M427
6993  LD      B25B
      AND     X46  ; Manual 'OFF'
      OR      B49  ; Mist OFF on GOT
      OUT     M435
6997  LD      B25D
      AND     X47  ; Manual 'ON'
      OR      B4C
      OR      M428  ; Coolant test On(Adjust)
      ANI     M436
      OUT     M428  ; Coolant test On(Adjust)
7003  LD      B25D
      AND     X46  ; Manual 'OFF'
      OR      B4D
      OUT     M436
7007  LD      B25C
      AND     X47  ; Manual 'ON'
      OR      B4A  ; Air Blow On on GOT
      OR      M429  ; Air Blow test On(Adjust)
      ANI     M437
      OUT     M429  ; Air Blow test On(Adjust)
7013  LD      B25C
      AND     X46  ; Manual 'OFF'
      OR      B4B  ; Air Blow Off on GOT
      OUT     M437
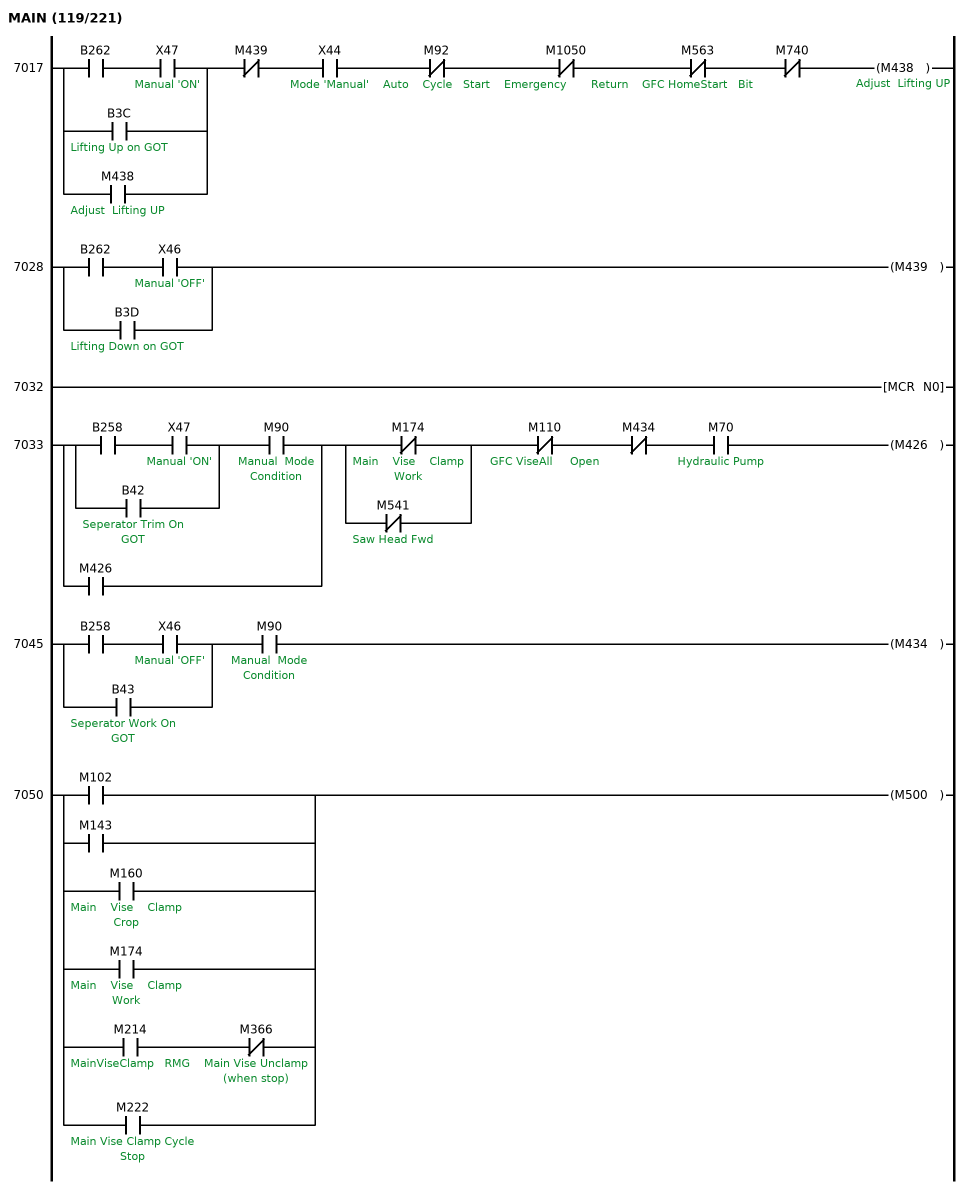
7017  LD      B262
      AND     X47  ; Manual 'ON'
      OR      B3C  ; Lifting Up on GOT
      OR      M438  ; Adjust  Lifting UP
      ANI     M439
      AND     X44  ; Mode 'Manual'
      ANI     M92  ; Auto    Cycle   Start
      ANI     M1050  ; Emergency       Return
      ANI     M563  ; GFC HomeStart   Bit
      ANI     M740
      OUT     M438  ; Adjust  Lifting UP
7028  LD      B262
      AND     X46  ; Manual 'OFF'
      OR      B3D  ; Lifting Down on GOT
      OUT     M439
7032  MCR     N0
7033  LD      B258
      AND     X47  ; Manual 'ON'
      OR      B42  ; Seperator Trim On GOT
      AND     M90  ; Manual  Mode    Condition
      OR      M426
      LDI     M174  ; Main    Vise    Clamp   Work
      ORI     M541  ; Saw Head Fwd
      ANB
      ANI     M110  ; GFC ViseAll     Open
      ANI     M434
      AND     M70  ; Hydraulic Pump
      OUT     M426
7045  LD      B258
      AND     X46  ; Manual 'OFF'
      OR      B43  ; Seperator Work On GOT
      AND     M90  ; Manual  Mode    Condition
      OUT     M434
7050  LD      M102
      OR      M143
      OR      M160  ; Main    Vise    Clamp   Crop
      OR      M174  ; Main    Vise    Clamp   Work
      LD      M214  ; MainViseClamp   RMG
      ANI     M366  ; Main Vise Unclamp (when stop)
      ORB
      OR      M222  ; Main Vise Clamp Cycle Stop
      OUT     M500
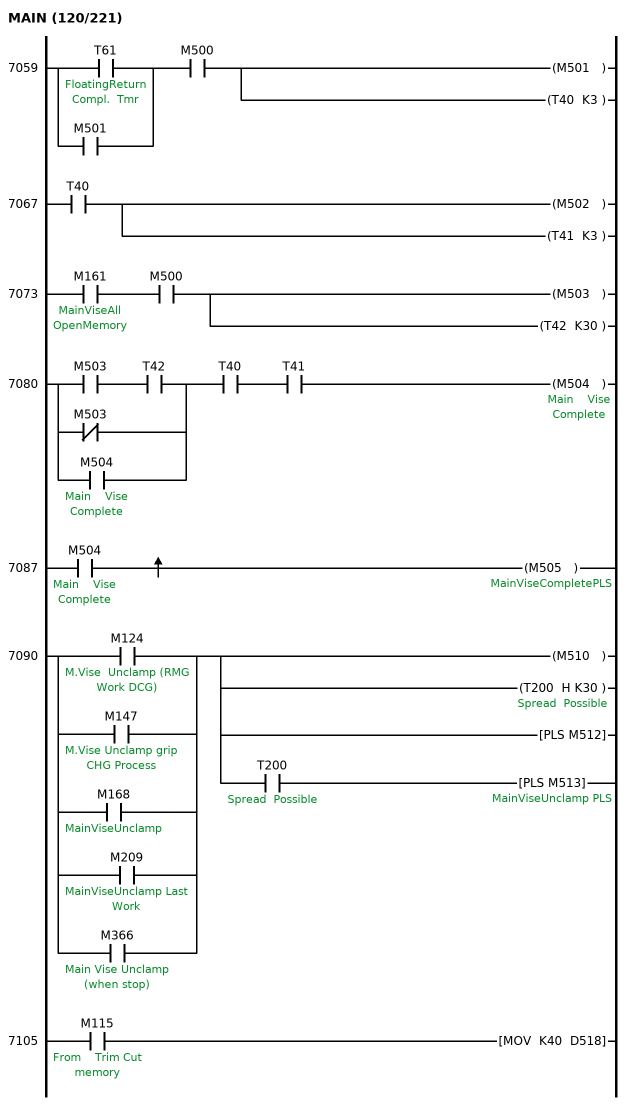
7059  LD      T61  ; FloatingReturn  Compl.  Tmr
      OR      M501
      AND     M500
      OUT     M501
      OUT     T40 K3
7067  LD      T40
      OUT     M502
      OUT     T41 K3
7073  LD      M161  ; MainViseAll OpenMemory
      AND     M500
      OUT     M503
      OUT     T42 K30
7080  LD      M503
      AND     T42
      ORI     M503
      OR      M504  ; Main    Vise    Complete
      AND     T40
      AND     T41
      OUT     M504  ; Main    Vise    Complete
7087  LD      M504  ; Main    Vise    Complete
      MEP
      OUT     M505  ; MainViseCompletePLS
7090  LD      M124  ; M.Vise  Unclamp (RMG Work DCG)
      OR      M147  ; M.Vise Unclamp grip CHG Process
      OR      M168  ; MainViseUnclamp
      OR      M209  ; MainViseUnclamp Last    Work
      OR      M366  ; Main Vise Unclamp (when stop)
      OUT     M510
      OUTH    T200 K30  ; Spread  Possible
      PLS     M512
      AND     T200  ; Spread  Possible
      PLS     M513  ; MainViseUnclamp PLS
7105  LD      M115  ; From    Trim Cut memory
      MOV     K40 D518
